C09091=1072.095,-108.990,-56.403,172.612,21.671,153.924
C09092=1072.101,-108.740,-56.412,172.614,21.673,153.924
C09093=1072.107,-108.490,-56.422,172.616,21.674,153.924
C09094=1072.114,-108.241,-56.432,172.617,21.675,153.924
C09095=1072.120,-107.991,-56.442,172.619,21.676,153.924
C09096=1072.126,-107.741,-56.451,172.621,21.677,153.924
C09097=1072.132,-107.492,-56.461,172.622,21.678,153.924
C09098=1072.138,-107.242,-56.470,172.624,21.680,153.924
C09099=1072.144,-106.992,-56.481,172.625,21.681,153.924
C09100=1072.150,-106.743,-56.491,172.626,21.681,153.924
C09101=1072.156,-106.493,-56.500,172.628,21.683,153.924
C09102=1072.162,-106.243,-56.510,172.629,21.684,153.924
C09103=1072.169,-105.993,-56.521,172.631,21.685,153.924
C09104=1072.175,-105.743,-56.531,172.633,21.686,153.924
C09105=1072.181,-105.493,-56.540,172.634,21.688,153.924
C09106=1072.187,-105.243,-56.550,172.636,21.689,153.924
C09107=1072.193,-104.994,-56.561,172.638,21.690,153.924
C09108=1072.199,-104.744,-56.570,172.639,21.691,153.924
C09109=1072.205,-104.494,-56.580,172.641,21.693,153.924
C09110=1072.212,-104.245,-56.589,172.643,21.694,153.924
C09111=1072.217,-103.995,-56.600,172.644,21.695,153.924
C09112=1072.223,-103.745,-56.610,172.646,21.696,153.924
C09113=1072.230,-103.495,-56.619,172.648,21.697,153.924
C09114=1072.236,-103.246,-56.630,172.649,21.699,153.924
C09115=1072.242,-102.996,-56.640,172.651,21.700,153.924
C09116=1072.248,-102.746,-56.649,172.652,21.701,153.924
C09117=1072.254,-102.497,-56.660,172.654,21.702,153.924
C09118=1072.260,-102.247,-56.670,172.656,21.704,153.924
C09119=1072.266,-101.997,-56.679,172.657,21.705,153.924
C09120=1072.272,-101.748,-56.690,172.659,21.706,153.924
C09121=1072.278,-101.498,-56.699,172.660,21.708,153.924
C09122=1072.284,-101.249,-56.710,172.662,21.709,153.924
C09123=1072.290,-100.999,-56.720,172.663,21.710,153.924
C09124=1072.297,-100.748,-56.730,172.664,21.711,153.924
C09125=1072.303,-100.499,-56.741,172.666,21.712,153.924
C09126=1072.309,-100.249,-56.750,172.668,21.714,153.924
C09127=1072.316,-100.000,-56.760,172.669,21.715,153.924
C09128=1072.321,-99.750,-56.771,172.671,21.716,153.924
C09129=1072.327,-99.500,-56.780,172.672,21.717,153.924
C09130=1072.334,-99.251,-56.790,172.674,21.719,153.924
C09131=1072.339,-99.001,-56.801,172.676,21.720,153.924
C09132=1072.346,-98.752,-56.811,172.677,21.721,153.924
C09133=1072.352,-98.501,-56.821,172.679,21.722,153.924
C09134=1072.359,-98.220,-56.833,172.681,21.724,153.924
C09135=1072.365,-97.938,-56.844,172.683,21.726,153.924
C09136=1072.373,-97.657,-56.855,172.685,21.727,153.924
C09137=1072.379,-97.374,-56.867,172.686,21.728,153.924
C09138=1072.386,-97.125,-56.877,172.688,21.730,153.924
C09139=1072.391,-96.875,-56.887,172.689,21.731,153.924
C09140=1072.397,-96.626,-56.898,172.691,21.733,153.924
C09141=1072.403,-96.376,-56.907,172.692,21.734,153.924
C09142=1072.409,-96.126,-56.918,172.694,21.735,153.924
C09143=1072.415,-95.877,-56.929,172.696,21.737,153.924
C09144=1072.421,-95.626,-56.939,172.697,21.738,153.924
C09145=1072.428,-95.377,-56.949,172.699,21.739,153.924
C09146=1072.433,-95.127,-56.960,172.700,21.741,153.924
C09147=1072.440,-94.878,-56.970,172.702,21.742,153.924
C09148=1072.445,-94.628,-56.980,172.703,21.744,153.924
C09149=1072.452,-94.379,-56.990,172.705,21.745,153.924
C09150=1072.457,-94.128,-57.000,172.707,21.746,153.924
C09151=1072.464,-93.879,-57.011,172.708,21.748,153.924
C09152=1072.470,-93.629,-57.022,172.710,21.749,153.924
C09153=1072.475,-93.379,-57.032,172.711,21.751,153.924
C09154=1072.482,-93.130,-57.042,172.713,21.753,153.924
C09155=1072.487,-92.880,-57.053,172.714,21.754,153.924
C09156=1072.494,-92.630,-57.063,172.716,21.755,153.924
C09157=1072.500,-92.381,-57.074,172.717,21.757,153.924
C09158=1072.506,-92.131,-57.083,172.719,21.758,153.924
C09159=1072.512,-91.881,-57.095,172.721,21.759,153.924
C09160=1072.518,-91.631,-57.105,172.722,21.761,153.924
C09161=1072.524,-91.382,-57.115,172.724,21.762,153.924
C09162=1072.530,-91.132,-57.126,172.725,21.764,153.924
C09163=1072.536,-90.882,-57.135,172.727,21.765,153.924
C09164=1072.542,-90.632,-57.147,172.728,21.766,153.924
C09165=1072.548,-90.383,-57.158,172.730,21.768,153.924
C09166=1072.554,-90.133,-57.167,172.731,21.770,153.924
C09167=1072.560,-89.883,-57.178,172.733,21.771,153.924
C09168=1072.566,-89.634,-57.188,172.735,21.773,153.924
C09169=1072.573,-89.384,-57.200,172.736,21.774,153.924
C09170=1072.578,-89.134,-57.210,172.738,21.775,153.924
C09171=1072.585,-88.885,-57.220,172.739,21.777,153.924
C09172=1072.590,-88.635,-57.231,172.741,21.778,153.924
C09173=1072.597,-88.386,-57.240,172.742,21.780,153.925
C09174=1072.603,-88.135,-57.252,172.744,21.781,153.925
C09175=1072.609,-87.886,-57.263,172.745,21.783,153.925
C09176=1072.615,-87.637,-57.273,172.747,21.784,153.925
C09177=1072.621,-87.387,-57.283,172.748,21.786,153.925
C09178=1072.628,-87.137,-57.294,172.750,21.787,153.925
C09179=1072.633,-86.887,-57.305,172.751,21.789,153.925
C09180=1072.639,-86.638,-57.315,172.753,21.790,153.925
C09181=1072.646,-86.389,-57.326,172.755,21.792,153.925
C09182=1072.652,-86.138,-57.336,172.756,21.793,153.925
C09183=1072.657,-85.888,-57.347,172.758,21.794,153.925
C09184=1072.664,-85.639,-57.357,172.759,21.796,153.925
C09185=1072.670,-85.389,-57.369,172.761,21.798,153.925
C09186=1072.676,-85.139,-57.380,172.762,21.799,153.925
C09187=1072.682,-84.890,-57.389,172.764,21.801,153.925
C09188=1072.688,-84.640,-57.400,172.765,21.802,153.925
C09189=1072.694,-84.390,-57.411,172.767,21.804,153.925
C09190=1072.701,-84.141,-57.421,172.768,21.805,153.925
C09191=1072.706,-83.891,-57.432,172.770,21.807,153.925
C09192=1072.713,-83.641,-57.444,172.772,21.808,153.925
C09193=1072.719,-83.392,-57.454,172.773,21.809,153.925
C09194=1072.725,-83.142,-57.464,172.774,21.811,153.926
C09195=1072.731,-82.892,-57.475,172.776,21.813,153.926
C09196=1072.737,-82.642,-57.486,172.778,21.814,153.926
C09197=1072.743,-82.393,-57.496,172.779,21.816,153.926
C09198=1072.750,-82.113,-57.508,172.781,21.817,153.926
C09199=1072.758,-81.834,-57.520,172.783,21.819,153.926
C09200=1072.764,-81.554,-57.533,172.784,21.821,153.926
C09201=1072.771,-81.275,-57.545,172.786,21.823,153.926
C09202=1072.777,-81.026,-57.556,172.788,21.824,153.926
C09203=1072.784,-80.776,-57.566,172.789,21.826,153.926
C09204=1072.790,-80.526,-57.577,172.791,21.827,153.926
C09205=1072.795,-80.277,-57.588,172.792,21.829,153.926
C09206=1072.802,-80.027,-57.599,172.793,21.831,153.926
C09207=1072.808,-79.778,-57.610,172.795,21.832,153.926
C09208=1072.814,-79.527,-57.620,172.797,21.833,153.926
C09209=1072.820,-79.277,-57.631,172.798,21.835,153.926
C09210=1072.826,-79.028,-57.642,172.800,21.837,153.926
C09211=1072.832,-78.778,-57.653,172.801,21.839,153.927
C09212=1072.838,-78.528,-57.664,172.803,21.840,153.927
C09213=1072.844,-78.279,-57.675,172.804,21.842,153.927
C09214=1072.850,-78.030,-57.687,172.805,21.843,153.927
C09215=1072.857,-77.780,-57.697,172.807,21.845,153.927
C09216=1072.862,-77.530,-57.708,172.809,21.847,153.927
C09217=1072.869,-77.280,-57.719,172.811,21.848,153.927
C09218=1072.875,-77.031,-57.730,172.812,21.850,153.927
C09219=1072.880,-76.781,-57.741,172.814,21.852,153.927
C09220=1072.887,-76.531,-57.752,172.815,21.854,153.927
C09221=1072.892,-76.281,-57.763,172.817,21.855,153.927
C09222=1072.898,-76.032,-57.774,172.818,21.857,153.927
C09223=1072.904,-75.782,-57.785,172.820,21.858,153.927
C09224=1072.910,-75.532,-57.796,172.821,21.860,153.928
C09225=1072.917,-75.282,-57.807,172.823,21.862,153.928
C09226=1072.923,-75.033,-57.818,172.824,21.864,153.928
C09227=1072.929,-74.783,-57.829,172.826,21.865,153.928
C09228=1072.935,-74.534,-57.841,172.827,21.867,153.928
C09229=1072.941,-74.284,-57.851,172.829,21.868,153.928
C09230=1072.947,-74.034,-57.863,172.830,21.870,153.928
C09231=1072.953,-73.785,-57.874,172.832,21.872,153.928
C09232=1072.959,-73.535,-57.884,172.833,21.874,153.928
C09233=1072.965,-73.285,-57.896,172.835,21.875,153.928
C09234=1072.970,-73.035,-57.907,172.836,21.877,153.928
C09235=1072.976,-72.786,-57.919,172.837,21.879,153.929
C09236=1072.983,-72.536,-57.930,172.839,21.880,153.929
C09237=1072.988,-72.287,-57.941,172.840,21.882,153.929
C09238=1072.994,-72.037,-57.952,172.842,21.884,153.929
C09239=1073.000,-71.787,-57.963,172.843,21.886,153.929
C09240=1073.007,-71.538,-57.975,172.845,21.888,153.929
C09241=1073.012,-71.288,-57.986,172.847,21.890,153.929
C09242=1073.018,-71.038,-57.997,172.848,21.891,153.929
C09243=1073.024,-70.789,-58.008,172.850,21.893,153.929
C09244=1073.030,-70.538,-58.019,172.851,21.895,153.930
C09245=1073.036,-70.290,-58.031,172.853,21.897,153.930
C09246=1073.042,-70.039,-58.042,172.854,21.898,153.930
C09247=1073.048,-69.790,-58.053,172.856,21.900,153.930
C09248=1073.053,-69.540,-58.065,172.857,21.902,153.930
C09249=1073.060,-69.291,-58.077,172.859,21.904,153.930
C09250=1073.065,-69.041,-58.087,172.860,21.906,153.930
C09251=1073.072,-68.791,-58.099,172.861,21.908,153.930
C09252=1073.078,-68.542,-58.110,172.863,21.909,153.930
C09253=1073.084,-68.292,-58.122,172.864,21.911,153.930
C09254=1073.089,-68.042,-58.133,172.866,21.913,153.931
C09255=1073.095,-67.792,-58.144,172.867,21.914,153.931
C09256=1073.102,-67.543,-58.156,172.869,21.916,153.931
C09257=1073.107,-67.293,-58.167,172.870,21.918,153.931
C09258=1073.114,-67.043,-58.178,172.871,21.920,153.931
C09259=1073.119,-66.794,-58.190,172.873,21.921,153.931
C09260=1073.125,-66.544,-58.201,172.875,21.924,153.931
C09261=1073.131,-66.295,-58.213,172.877,21.926,153.931
C09262=1073.138,-66.018,-58.226,172.878,21.928,153.932
C09263=1073.145,-65.740,-58.238,172.879,21.930,153.932
C09264=1073.152,-65.463,-58.250,172.881,21.931,153.932
C09265=1073.158,-65.185,-58.264,172.883,21.934,153.932
C09266=1073.164,-64.937,-58.275,172.885,21.935,153.932
C09267=1073.170,-64.686,-58.286,172.886,21.937,153.932
C09268=1073.176,-64.438,-58.298,172.887,21.939,153.932
C09269=1073.182,-64.187,-58.310,172.889,21.941,153.932
C09270=1073.188,-63.937,-58.321,172.890,21.943,153.933
C09271=1073.194,-63.688,-58.333,172.892,21.944,153.933
C09272=1073.200,-63.438,-58.344,172.893,21.946,153.933
C09273=1073.206,-63.189,-58.356,172.895,21.948,153.933
C09274=1073.212,-62.938,-58.367,172.896,21.950,153.933
C09275=1073.218,-62.689,-58.379,172.897,21.952,153.933
C09276=1073.224,-62.439,-58.390,172.899,21.953,153.933
C09277=1073.230,-62.190,-58.402,172.900,21.955,153.933
C09278=1073.236,-61.940,-58.414,172.903,21.958,153.933
C09279=1073.242,-61.691,-58.425,172.904,21.960,153.934
C09280=1073.248,-61.441,-58.436,172.905,21.962,153.934
C09281=1073.254,-61.192,-58.448,172.907,21.963,153.934
C09282=1073.260,-60.941,-58.460,172.908,21.965,153.934
C09283=1073.267,-60.692,-58.472,172.910,21.967,153.934
C09284=1073.272,-60.442,-58.483,172.911,21.969,153.934
C09285=1073.279,-60.193,-58.495,172.912,21.971,153.934
C09286=1073.284,-59.943,-58.506,172.914,21.973,153.935
C09287=1073.291,-59.693,-58.518,172.915,21.974,153.935
C09288=1073.297,-59.443,-58.529,172.917,21.976,153.935
C09289=1073.302,-59.194,-58.542,172.918,21.978,153.935
C09290=1073.309,-58.944,-58.553,172.920,21.980,153.935
C09291=1073.315,-58.695,-58.564,172.921,21.982,153.935
C09292=1073.321,-58.445,-58.576,172.923,21.984,153.935
C09293=1073.327,-58.195,-58.588,172.925,21.986,153.935
C09294=1073.333,-57.946,-58.600,172.926,21.987,153.935
C09295=1073.339,-57.696,-58.611,172.928,21.989,153.936
C09296=1073.345,-57.446,-58.624,172.929,21.991,153.936
C09297=1073.351,-57.197,-58.635,172.930,21.993,153.936
C09298=1073.358,-56.947,-58.646,172.932,21.995,153.936
C09299=1073.363,-56.698,-58.659,172.933,21.997,153.936
C09300=1073.369,-56.448,-58.670,172.935,21.999,153.936
C09301=1073.376,-56.198,-58.682,172.936,22.001,153.937
C09302=1073.382,-55.949,-58.693,172.937,22.002,153.937
C09303=1073.388,-55.699,-58.705,172.939,22.004,153.937
C09304=1073.394,-55.449,-58.717,172.940,22.006,153.937
C09305=1073.400,-55.200,-58.729,172.942,22.008,153.937
C09306=1073.406,-54.950,-58.741,172.944,22.010,153.937
C09307=1073.413,-54.700,-58.753,172.945,22.012,153.937
C09308=1073.419,-54.451,-58.764,172.947,22.014,153.937
C09309=1073.425,-54.201,-58.777,172.948,22.016,153.938
C09310=1073.431,-53.951,-58.788,172.949,22.018,153.938
C09311=1073.438,-53.702,-58.800,172.951,22.020,153.938
C09312=1073.443,-53.452,-58.812,172.952,22.022,153.938
C09313=1073.449,-53.202,-58.823,172.954,22.024,153.938
C09314=1073.456,-52.953,-58.835,172.955,22.025,153.938
C09315=1073.461,-52.703,-58.847,172.957,22.027,153.938
C09316=1073.468,-52.454,-58.859,172.958,22.029,153.939
C09317=1073.473,-52.203,-58.871,172.959,22.031,153.939
C09318=1073.480,-51.954,-58.883,172.962,22.033,153.939
C09319=1073.486,-51.705,-58.895,172.963,22.035,153.939
C09320=1073.492,-51.455,-58.907,172.964,22.037,153.939
C09321=1073.499,-51.206,-58.919,172.966,22.039,153.939
C09322=1073.505,-50.955,-58.931,172.967,22.041,153.939
C09323=1073.510,-50.706,-58.943,172.969,22.043,153.940
C09324=1073.517,-50.457,-58.955,172.970,22.045,153.940
C09325=1073.523,-50.207,-58.967,172.971,22.047,153.940
C09326=1073.529,-49.931,-58.980,172.973,22.049,153.940
C09327=1073.536,-49.655,-58.994,172.975,22.052,153.940
C09328=1073.543,-49.379,-59.007,172.976,22.054,153.940
C09329=1073.549,-49.103,-59.021,172.978,22.056,153.941
C09330=1073.555,-48.854,-59.033,172.979,22.058,153.941
C09331=1073.561,-48.604,-59.044,172.981,22.060,153.941
C09332=1073.567,-48.354,-59.056,172.983,22.062,153.941
C09333=1073.573,-48.105,-59.069,172.984,22.064,153.941
C09334=1073.579,-47.855,-59.081,172.985,22.066,153.941
C09335=1073.585,-47.605,-59.093,172.987,22.068,153.942
C09336=1073.591,-47.356,-59.106,172.988,22.070,153.942
C09337=1073.597,-47.106,-59.118,172.989,22.072,153.942
C09338=1073.603,-46.857,-59.130,172.991,22.074,153.942
C09339=1073.609,-46.607,-59.142,172.992,22.076,153.942
C09340=1073.614,-46.358,-59.155,172.993,22.078,153.942
C09341=1073.621,-46.108,-59.167,172.995,22.080,153.943
C09342=1073.627,-45.858,-59.179,172.997,22.083,153.943
C09343=1073.633,-45.608,-59.191,172.998,22.085,153.943
C09344=1073.639,-45.359,-59.203,173.000,22.087,153.943
C09345=1073.644,-45.109,-59.215,173.001,22.089,153.943
C09346=1073.650,-44.859,-59.228,173.003,22.091,153.943
C09347=1073.657,-44.610,-59.240,173.004,22.093,153.944
C09348=1073.662,-44.360,-59.252,173.005,22.095,153.944
C09349=1073.668,-44.111,-59.264,173.007,22.097,153.944
C09350=1073.675,-43.861,-59.276,173.008,22.099,153.944
C09351=1073.681,-43.611,-59.289,173.009,22.101,153.944
C09352=1073.687,-43.361,-59.301,173.012,22.103,153.944
C09353=1073.692,-43.112,-59.314,173.013,22.106,153.945
C09354=1073.699,-42.862,-59.326,173.014,22.108,153.945
C09355=1073.705,-42.613,-59.339,173.016,22.110,153.945
C09356=1073.711,-42.363,-59.351,173.017,22.112,153.945
C09357=1073.717,-42.114,-59.363,173.018,22.113,153.945
C09358=1073.723,-41.865,-59.376,173.020,22.116,153.946
C09359=1073.729,-41.615,-59.388,173.021,22.118,153.946
C09360=1073.735,-41.365,-59.401,173.022,22.120,153.946
C09361=1073.741,-41.115,-59.413,173.024,22.122,153.946
C09362=1073.747,-40.865,-59.425,173.026,22.124,153.946
C09363=1073.752,-40.616,-59.437,173.027,22.126,153.947
C09364=1073.759,-40.367,-59.449,173.029,22.128,153.947
C09365=1073.765,-40.117,-59.462,173.030,22.130,153.947
C09366=1073.771,-39.867,-59.475,173.031,22.132,153.947
C09367=1073.777,-39.618,-59.488,173.033,22.135,153.947
C09368=1073.784,-39.368,-59.500,173.034,22.137,153.947
C09369=1073.790,-39.118,-59.512,173.035,22.139,153.948
C09370=1073.795,-38.869,-59.524,173.037,22.140,153.948
C09371=1073.801,-38.619,-59.537,173.038,22.143,153.948
C09372=1073.807,-38.369,-59.549,173.040,22.145,153.948
C09373=1073.814,-38.120,-59.562,173.042,22.147,153.948
C09374=1073.820,-37.870,-59.575,173.043,22.150,153.949
C09375=1073.826,-37.620,-59.587,173.044,22.152,153.949
C09376=1073.831,-37.371,-59.599,173.046,22.154,153.949
C09377=1073.837,-37.121,-59.612,173.047,22.156,153.949
C09378=1073.843,-36.872,-59.625,173.048,22.158,153.949
C09379=1073.849,-36.622,-59.638,173.050,22.160,153.949
C09380=1073.855,-36.372,-59.650,173.051,22.162,153.950
C09381=1073.861,-36.122,-59.663,173.053,22.165,153.950
C09382=1073.866,-35.873,-59.675,173.054,22.167,153.950
C09383=1073.872,-35.624,-59.688,173.056,22.169,153.950
C09384=1073.878,-35.374,-59.701,173.057,22.171,153.950
C09385=1073.884,-35.124,-59.713,173.058,22.173,153.951
C09386=1073.890,-34.875,-59.727,173.060,22.175,153.951
C09387=1073.896,-34.625,-59.739,173.061,22.177,153.951
C09388=1073.903,-34.375,-59.751,173.062,22.180,153.951
C09389=1073.909,-34.126,-59.764,173.064,22.182,153.951
C09390=1073.915,-33.851,-59.779,173.066,22.185,153.952
C09391=1073.922,-33.575,-59.792,173.067,22.186,153.952
C09392=1073.928,-33.300,-59.806,173.068,22.189,153.952
C09393=1073.935,-33.024,-59.820,173.071,22.192,153.952
C09394=1073.941,-32.775,-59.833,173.072,22.194,153.953
C09395=1073.947,-32.525,-59.846,173.073,22.196,153.953
C09396=1073.953,-32.275,-59.858,173.075,22.198,153.953
C09397=1073.959,-32.026,-59.872,173.076,22.200,153.953
C09398=1073.965,-31.776,-59.884,173.077,22.203,153.953
C09399=1073.971,-31.526,-59.897,173.079,22.204,153.954
C09400=1073.977,-31.277,-59.910,173.081,22.207,153.954
C09401=1073.983,-31.027,-59.923,173.082,22.209,153.954
C09402=1073.989,-30.777,-59.935,173.083,22.211,153.954
C09403=1073.995,-30.528,-59.948,173.085,22.214,153.954
C09404=1074.001,-30.278,-59.961,173.086,22.216,153.955
C09405=1074.007,-30.029,-59.974,173.087,22.218,153.955
C09406=1074.013,-29.779,-59.987,173.089,22.220,153.955
C09407=1074.019,-29.530,-60.000,173.090,22.222,153.955
C09408=1074.024,-29.280,-60.012,173.091,22.224,153.955
C09409=1074.030,-29.030,-60.025,173.094,22.227,153.956
C09410=1074.037,-28.781,-60.038,173.095,22.229,153.956
C09411=1074.042,-28.531,-60.051,173.096,22.231,153.956
C09412=1074.049,-28.282,-60.064,173.097,22.233,153.956
C09413=1074.055,-28.032,-60.076,173.099,22.235,153.956
C09414=1074.061,-27.783,-60.090,173.100,22.238,153.957
C09415=1074.067,-27.533,-60.102,173.101,22.240,153.957
C09416=1074.073,-27.284,-60.115,173.103,22.242,153.957
C09417=1074.079,-27.034,-60.128,173.104,22.244,153.957
C09418=1074.084,-26.784,-60.142,173.106,22.246,153.957
C09419=1074.090,-26.534,-60.154,173.108,22.249,153.958
C09420=1074.096,-26.285,-60.168,173.109,22.251,153.958
C09421=1074.102,-26.035,-60.180,173.110,22.253,153.958
C09422=1074.109,-25.786,-60.194,173.111,22.256,153.958
C09423=1074.114,-25.536,-60.207,173.113,22.258,153.959
C09424=1074.120,-25.287,-60.220,173.114,22.260,153.959
C09425=1074.126,-25.037,-60.233,173.115,22.262,153.959
C09426=1074.132,-24.787,-60.246,173.117,22.265,153.959
C09427=1074.138,-24.538,-60.260,173.119,22.267,153.959
C09428=1074.143,-24.288,-60.272,173.120,22.269,153.960
C09429=1074.150,-24.039,-60.285,173.121,22.272,153.960
C09430=1074.156,-23.789,-60.299,173.123,22.274,153.960
C09431=1074.162,-23.540,-60.311,173.124,22.276,153.960
C09432=1074.167,-23.290,-60.325,173.125,22.278,153.961
C09433=1074.173,-23.040,-60.338,173.127,22.281,153.961
C09434=1074.179,-22.791,-60.351,173.129,22.283,153.961
C09435=1074.186,-22.542,-60.364,173.130,22.285,153.961
C09436=1074.191,-22.291,-60.377,173.131,22.288,153.962
C09437=1074.197,-22.042,-60.391,173.133,22.290,153.962
C09438=1074.203,-21.793,-60.404,173.134,22.292,153.962
C09439=1074.208,-21.543,-60.417,173.135,22.294,153.962
C09440=1074.215,-21.293,-60.431,173.137,22.297,153.963
C09441=1074.221,-21.043,-60.444,173.138,22.298,153.963
C09442=1074.227,-20.794,-60.457,173.140,22.301,153.963
C09443=1074.233,-20.544,-60.470,173.141,22.304,153.963
C09444=1074.239,-20.295,-60.484,173.143,22.306,153.963
C09445=1074.245,-20.045,-60.496,173.144,22.308,153.964
C09446=1074.251,-19.796,-60.509,173.145,22.310,153.964
C09447=1074.257,-19.546,-60.523,173.146,22.313,153.964
C09448=1074.263,-19.297,-60.537,173.148,22.315,153.964
C09449=1074.269,-19.047,-60.549,173.149,22.317,153.965
C09450=1074.274,-18.797,-60.563,173.151,22.320,153.965
C09451=1074.280,-18.548,-60.576,173.153,22.322,153.965
C09452=1074.287,-18.299,-60.590,173.154,22.324,153.965
C09453=1074.292,-18.048,-60.603,173.155,22.327,153.965
C09454=1074.299,-17.772,-60.618,173.156,22.329,153.966
C09455=1074.306,-17.496,-60.633,173.159,22.331,153.966
C09456=1074.313,-17.219,-60.647,173.160,22.334,153.966
C09457=1074.319,-16.943,-60.662,173.161,22.336,153.966
C09458=1074.325,-16.694,-60.675,173.162,22.339,153.967
C09459=1074.331,-16.444,-60.689,173.165,22.341,153.967
C09460=1074.337,-16.195,-60.702,173.166,22.344,153.967
C09461=1074.343,-15.946,-60.716,173.167,22.346,153.967
C09462=1074.349,-15.695,-60.730,173.168,22.348,153.968
C09463=1074.355,-15.445,-60.742,173.170,22.350,153.968
C09464=1074.362,-15.196,-60.756,173.171,22.352,153.968
C09465=1074.367,-14.947,-60.769,173.172,22.355,153.968
C09466=1074.373,-14.697,-60.783,173.174,22.358,153.969
C09467=1074.379,-14.448,-60.797,173.176,22.360,153.969
C09468=1074.385,-14.198,-60.810,173.177,22.362,153.969
C09469=1074.390,-13.949,-60.824,173.178,22.364,153.969
C09470=1074.397,-13.699,-60.837,173.179,22.367,153.970
C09471=1074.403,-13.449,-60.851,173.181,22.369,153.970
C09472=1074.409,-13.199,-60.864,173.182,22.371,153.970
C09473=1074.414,-12.950,-60.878,173.183,22.374,153.970
C09474=1074.420,-12.701,-60.891,173.185,22.377,153.971
C09475=1074.426,-12.451,-60.905,173.187,22.379,153.971
C09476=1074.432,-12.202,-60.918,173.188,22.381,153.971
C09477=1074.438,-11.952,-60.932,173.189,22.383,153.971
C09478=1074.444,-11.702,-60.946,173.191,22.385,153.971
C09479=1074.450,-11.453,-60.959,173.192,22.388,153.972
C09480=1074.455,-11.203,-60.973,173.193,22.390,153.972
C09481=1074.461,-10.954,-60.987,173.195,22.393,153.972
C09482=1074.467,-10.704,-61.000,173.197,22.395,153.972
C09483=1074.474,-10.454,-61.014,173.198,22.397,153.973
C09484=1074.479,-10.205,-61.028,173.199,22.400,153.973
C09485=1074.485,-9.955,-61.041,173.200,22.402,153.973
C09486=1074.491,-9.706,-61.055,173.202,22.404,153.973
C09487=1074.497,-9.457,-61.068,173.203,22.407,153.974
C09488=1074.503,-9.206,-61.083,173.204,22.409,153.974
C09489=1074.509,-8.957,-61.096,173.206,22.412,153.974
C09490=1074.515,-8.708,-61.110,173.208,22.414,153.974
C09491=1074.520,-8.458,-61.124,173.209,22.416,153.975
C09492=1074.527,-8.209,-61.137,173.210,22.419,153.975
C09493=1074.533,-7.959,-61.152,173.211,22.421,153.975
C09494=1074.539,-7.710,-61.165,173.213,22.423,153.975
C09495=1074.545,-7.460,-61.179,173.214,22.426,153.976
C09496=1074.550,-7.211,-61.193,173.216,22.429,153.976
C09497=1074.557,-6.961,-61.206,173.217,22.431,153.976
C09498=1074.562,-6.711,-61.220,173.219,22.433,153.976
C09499=1074.569,-6.462,-61.234,173.220,22.435,153.977
C09500=1074.574,-6.212,-61.247,173.221,22.438,153.977
C09501=1074.580,-5.962,-61.262,173.223,22.440,153.977
C09502=1074.587,-5.713,-61.276,173.224,22.442,153.977
C09503=1074.592,-5.464,-61.289,173.226,22.445,153.978
C09504=1074.598,-5.214,-61.303,173.227,22.447,153.978
C09505=1074.604,-4.964,-61.317,173.228,22.449,153.978
C09506=1074.610,-4.715,-61.331,173.230,22.452,153.978
C09507=1074.616,-4.465,-61.344,173.231,22.454,153.979
C09508=1074.623,-4.216,-61.359,173.232,22.457,153.979
C09509=1074.629,-3.966,-61.372,173.234,22.459,153.979
C09510=1074.634,-3.717,-61.386,173.236,22.461,153.979
C09511=1074.640,-3.467,-61.400,173.237,22.464,153.980
C09512=1074.647,-3.217,-61.414,173.238,22.466,153.980
C09513=1074.652,-2.968,-61.428,173.239,22.469,153.980
C09514=1074.658,-2.719,-61.442,173.241,22.471,153.981
C09515=1074.664,-2.468,-61.456,173.242,22.473,153.981
C09516=1074.669,-2.219,-61.470,173.243,22.476,153.981
C09517=1074.675,-1.970,-61.485,173.245,22.479,153.981
C09518=1074.681,-1.692,-61.500,173.247,22.481,153.982
C09519=1074.688,-1.414,-61.515,173.248,22.484,153.982
C09520=1074.694,-1.136,-61.531,173.250,22.487,153.982
C09521=1074.701,-0.858,-61.547,173.251,22.489,153.982
C09522=1074.707,-0.608,-61.561,173.252,22.492,153.983
C09523=1074.712,-0.359,-61.576,173.253,22.494,153.983
C09524=1074.719,-0.109,-61.589,173.256,22.497,153.983
C09525=1074.725,0.140,-61.603,173.257,22.499,153.984
C09526=1074.730,0.390,-61.617,173.258,22.502,153.984
C09527=1074.737,0.639,-61.632,173.259,22.504,153.984
C09528=1074.742,0.889,-61.646,173.261,22.506,153.984
C09529=1074.748,1.138,-61.661,173.262,22.509,153.985
C09530=1074.753,1.387,-61.674,173.263,22.511,153.985
C09531=1074.759,1.638,-61.689,173.265,22.514,153.985
C09532=1074.765,1.887,-61.703,173.266,22.516,153.985
C09533=1074.771,2.136,-61.717,173.268,22.519,153.986
C09534=1074.777,2.386,-61.731,173.269,22.521,153.986
C09535=1074.783,2.635,-61.745,173.270,22.524,153.986
C09536=1074.789,2.885,-61.759,173.272,22.526,153.986
C09537=1074.795,3.134,-61.774,173.273,22.528,153.987
C09538=1074.801,3.384,-61.788,173.275,22.531,153.987
C09539=1074.806,3.633,-61.803,173.276,22.533,153.987
C09540=1074.812,3.883,-61.817,173.277,22.536,153.988
C09541=1074.818,4.133,-61.831,173.279,22.538,153.988
C09542=1074.824,4.382,-61.845,173.280,22.541,153.988
C09543=1074.830,4.632,-61.859,173.281,22.543,153.988
C09544=1074.836,4.881,-61.874,173.282,22.546,153.989
C09545=1074.842,5.131,-61.888,173.284,22.549,153.989
C09546=1074.847,5.380,-61.903,173.286,22.550,153.989
C09547=1074.854,5.629,-61.916,173.287,22.553,153.989
C09548=1074.860,5.879,-61.931,173.288,22.555,153.990
C09549=1074.866,6.129,-61.945,173.290,22.558,153.990
C09550=1074.872,6.378,-61.960,173.291,22.560,153.990
C09551=1074.877,6.628,-61.974,173.293,22.563,153.991
C09552=1074.883,6.877,-61.988,173.294,22.566,153.991
C09553=1074.889,7.127,-62.003,173.295,22.568,153.991
C09554=1074.895,7.376,-62.017,173.297,22.570,153.991
C09555=1074.901,7.626,-62.031,173.298,22.572,153.992
C09556=1074.907,7.875,-62.046,173.299,22.575,153.992
C09557=1074.913,8.124,-62.060,173.301,22.577,153.992
C09558=1074.919,8.375,-62.075,173.303,22.580,153.992
C09559=1074.925,8.624,-62.089,173.304,22.582,153.993
C09560=1074.931,8.874,-62.104,173.305,22.585,153.993
C09561=1074.936,9.123,-62.118,173.306,22.587,153.993
C09562=1074.943,9.372,-62.133,173.308,22.590,153.994
C09563=1074.948,9.622,-62.147,173.309,22.592,153.994
C09564=1074.955,9.872,-62.162,173.310,22.594,153.994
C09565=1074.960,10.121,-62.176,173.312,22.597,153.994
C09566=1074.966,10.371,-62.191,173.314,22.599,153.994
C09567=1074.972,10.620,-62.205,173.315,22.602,153.995
C09568=1074.978,10.870,-62.219,173.316,22.604,153.995
C09569=1074.984,11.119,-62.234,173.317,22.607,153.995
C09570=1074.990,11.369,-62.249,173.319,22.609,153.996
C09571=1074.996,11.618,-62.263,173.321,22.612,153.996
C09572=1075.002,11.868,-62.278,173.322,22.615,153.996
C09573=1075.008,12.117,-62.292,173.323,22.616,153.996
C09574=1075.014,12.367,-62.307,173.325,22.619,153.997
C09575=1075.020,12.616,-62.321,173.326,22.621,153.997
C09576=1075.026,12.866,-62.336,173.327,22.624,153.997
C09577=1075.032,13.115,-62.351,173.329,22.627,153.997
C09578=1075.038,13.365,-62.365,173.330,22.629,153.998
C09579=1075.044,13.614,-62.380,173.332,22.631,153.998
C09580=1075.050,13.864,-62.394,173.333,22.634,153.998
C09581=1075.056,14.113,-62.409,173.334,22.636,153.998
C09582=1075.063,14.393,-62.426,173.336,22.639,153.999
C09583=1075.069,14.673,-62.442,173.338,22.642,153.999
C09584=1075.076,14.953,-62.458,173.339,22.644,153.999
C09585=1075.082,15.233,-62.475,173.341,22.647,154.000
C09586=1075.088,15.483,-62.490,173.342,22.650,154.000
C09587=1075.094,15.732,-62.504,173.343,22.652,154.000
C09588=1075.100,15.981,-62.519,173.344,22.655,154.001
C09589=1075.106,16.230,-62.534,173.346,22.657,154.001
C09590=1075.112,16.481,-62.549,173.348,22.660,154.001
C09591=1075.117,16.730,-62.563,173.349,22.662,154.002
C09592=1075.124,16.979,-62.578,173.350,22.665,154.002
C09593=1075.129,17.228,-62.593,173.352,22.667,154.002
C09594=1075.135,17.478,-62.608,173.353,22.670,154.002
C09595=1075.141,17.727,-62.623,173.354,22.672,154.003
C09596=1075.147,17.977,-62.638,173.356,22.675,154.003
C09597=1075.153,18.227,-62.652,173.358,22.677,154.003
C09598=1075.158,18.477,-62.667,173.359,22.679,154.003
C09599=1075.165,18.726,-62.682,173.360,22.682,154.004
C09600=1075.171,18.975,-62.697,173.361,22.684,154.004
C09601=1075.177,19.225,-62.712,173.363,22.687,154.004
C09602=1075.182,19.474,-62.727,173.365,22.690,154.004
C09603=1075.188,19.724,-62.742,173.366,22.692,154.005
C09604=1075.194,19.973,-62.757,173.367,22.694,154.005
C09605=1075.200,20.223,-62.772,173.368,22.697,154.005
C09606=1075.206,20.472,-62.787,173.370,22.699,154.006
C09607=1075.212,20.721,-62.802,173.371,22.702,154.006
C09608=1075.218,20.971,-62.817,173.373,22.705,154.006
C09609=1075.223,21.220,-62.832,173.374,22.707,154.006
C09610=1075.230,21.470,-62.847,173.376,22.709,154.007
C09611=1075.235,21.719,-62.862,173.377,22.712,154.007
C09612=1075.241,21.969,-62.877,173.378,22.714,154.007
C09613=1075.247,22.219,-62.892,173.379,22.717,154.008
C09614=1075.253,22.468,-62.907,173.381,22.720,154.008
C09615=1075.259,22.717,-62.922,173.383,22.722,154.008
C09616=1075.264,22.967,-62.937,173.384,22.724,154.008
C09617=1075.270,23.216,-62.952,173.385,22.727,154.009
C09618=1075.277,23.466,-62.967,173.386,22.729,154.009
C09619=1075.282,23.715,-62.982,173.388,22.732,154.009
C09620=1075.288,23.965,-62.997,173.390,22.735,154.010
C09621=1075.293,24.214,-63.012,173.391,22.737,154.010
C09622=1075.300,24.464,-63.027,173.392,22.739,154.010
C09623=1075.305,24.714,-63.043,173.394,22.742,154.010
C09624=1075.311,24.963,-63.057,173.395,22.744,154.011
C09625=1075.317,25.212,-63.072,173.397,22.747,154.011
C09626=1075.323,25.462,-63.088,173.398,22.750,154.011
C09627=1075.329,25.711,-63.103,173.399,22.752,154.012
C09628=1075.335,25.961,-63.119,173.401,22.754,154.012
C09629=1075.341,26.210,-63.134,173.402,22.757,154.012
C09630=1075.347,26.459,-63.148,173.403,22.759,154.012
C09631=1075.353,26.709,-63.164,173.405,22.762,154.013
C09632=1075.359,26.959,-63.179,173.407,22.765,154.013
C09633=1075.364,27.208,-63.194,173.408,22.767,154.013
C09634=1075.371,27.457,-63.210,173.409,22.769,154.014
C09635=1075.376,27.707,-63.225,173.410,22.772,154.014
C09636=1075.382,27.956,-63.240,173.412,22.774,154.014
C09637=1075.388,28.206,-63.255,173.414,22.777,154.014
C09638=1075.394,28.456,-63.270,173.415,22.780,154.015
C09639=1075.400,28.704,-63.286,173.416,22.782,154.015
C09640=1075.406,28.954,-63.301,173.417,22.784,154.015
C09641=1075.412,29.204,-63.317,173.418,22.787,154.016
C09642=1075.417,29.453,-63.332,173.421,22.790,154.016
C09643=1075.423,29.702,-63.347,173.422,22.793,154.016
C09644=1075.429,29.952,-63.363,173.423,22.795,154.016
C09645=1075.435,30.201,-63.377,173.424,22.798,154.017
C09646=1075.441,30.483,-63.395,173.427,22.800,154.017
C09647=1075.448,30.764,-63.413,173.428,22.803,154.017
C09648=1075.455,31.045,-63.430,173.429,22.806,154.018
C09649=1075.460,31.326,-63.448,173.431,22.809,154.018
C09650=1075.467,31.576,-63.463,173.432,22.812,154.018
C09651=1075.473,31.826,-63.478,173.433,22.814,154.019
C09652=1075.479,32.075,-63.494,173.435,22.816,154.019
C09653=1075.484,32.324,-63.509,173.437,22.819,154.019
C09654=1075.490,32.574,-63.524,173.438,22.822,154.020
C09655=1075.497,32.823,-63.540,173.439,22.824,154.020
C09656=1075.502,33.073,-63.555,173.440,22.827,154.020
C09657=1075.507,33.323,-63.571,173.442,22.829,154.020
C09658=1075.514,33.572,-63.586,173.444,22.832,154.021
C09659=1075.520,33.822,-63.602,173.445,22.834,154.021
C09660=1075.525,34.070,-63.618,173.446,22.837,154.021
C09661=1075.531,34.320,-63.633,173.448,22.839,154.022
C09662=1075.537,34.570,-63.648,173.449,22.842,154.022
C09663=1075.543,34.819,-63.665,173.451,22.844,154.022
C09664=1075.549,35.068,-63.679,173.452,22.847,154.022
C09665=1075.555,35.318,-63.695,173.454,22.849,154.023
C09666=1075.560,35.568,-63.711,173.455,22.852,154.023
C09667=1075.567,35.817,-63.726,173.456,22.854,154.023
C09668=1075.572,36.066,-63.742,173.458,22.857,154.023
C09669=1075.578,36.316,-63.757,173.459,22.859,154.024
C09670=1075.584,36.565,-63.773,173.461,22.862,154.024
C09671=1075.590,36.815,-63.789,173.462,22.864,154.024
C09672=1075.596,37.064,-63.805,173.463,22.867,154.025
C09673=1075.601,37.313,-63.820,173.464,22.869,154.025
C09674=1075.608,37.562,-63.836,173.467,22.872,154.025
C09675=1075.613,37.812,-63.851,173.468,22.874,154.025
C09676=1075.619,38.062,-63.868,173.469,22.877,154.026
C09677=1075.625,38.312,-63.883,173.470,22.880,154.026
C09678=1075.631,38.560,-63.898,173.471,22.882,154.026
C09679=1075.637,38.810,-63.914,173.474,22.885,154.027
C09680=1075.643,39.059,-63.930,173.475,22.887,154.027
C09681=1075.648,39.309,-63.946,173.476,22.890,154.027
C09682=1075.654,39.559,-63.962,173.477,22.892,154.028
C09683=1075.659,39.808,-63.977,173.479,22.895,154.028
C09684=1075.665,40.057,-63.993,173.481,22.897,154.028
C09685=1075.672,40.306,-64.009,173.482,22.900,154.028
C09686=1075.678,40.556,-64.025,173.483,22.902,154.029
C09687=1075.683,40.806,-64.041,173.485,22.905,154.029
C09688=1075.689,41.055,-64.056,173.486,22.908,154.029
C09689=1075.694,41.304,-64.072,173.488,22.910,154.030
C09690=1075.700,41.554,-64.089,173.489,22.913,154.030
C09691=1075.706,41.804,-64.104,173.490,22.915,154.030
C09692=1075.712,42.053,-64.120,173.492,22.918,154.031
C09693=1075.718,42.302,-64.137,173.493,22.920,154.031
C09694=1075.724,42.551,-64.151,173.495,22.923,154.031
C09695=1075.730,42.801,-64.167,173.496,22.925,154.031
C09696=1075.735,43.051,-64.183,173.498,22.928,154.032
C09697=1075.741,43.300,-64.199,173.499,22.930,154.032
C09698=1075.747,43.549,-64.215,173.500,22.933,154.032
C09699=1075.753,43.799,-64.232,173.502,22.936,154.032
C09700=1075.759,44.049,-64.247,173.503,22.938,154.033
C09701=1075.764,44.297,-64.263,173.505,22.941,154.033
C09702=1075.770,44.547,-64.279,173.506,22.943,154.033
C09703=1075.776,44.797,-64.295,173.508,22.946,154.034
C09704=1075.782,45.046,-64.311,173.509,22.949,154.034
C09705=1075.788,45.295,-64.327,173.511,22.951,154.034
C09706=1075.792,45.544,-64.344,173.512,22.953,154.035
C09707=1075.798,45.794,-64.359,173.513,22.956,154.035
C09708=1075.804,46.044,-64.376,173.515,22.959,154.035
C09709=1075.810,46.293,-64.392,173.516,22.962,154.036
C09710=1075.816,46.575,-64.410,173.518,22.964,154.036
C09711=1075.822,46.855,-64.428,173.520,22.967,154.036
C09712=1075.829,47.137,-64.446,173.521,22.970,154.037
C09713=1075.836,47.418,-64.465,173.523,22.973,154.037
C09714=1075.841,47.668,-64.481,173.524,22.976,154.037
C09715=1075.847,47.918,-64.497,173.525,22.978,154.037
C09716=1075.853,48.167,-64.513,173.527,22.980,154.038
C09717=1075.858,48.415,-64.529,173.529,22.983,154.038
C09718=1075.864,48.665,-64.545,173.530,22.986,154.038
C09719=1075.870,48.914,-64.562,173.531,22.989,154.039
C09720=1075.876,49.164,-64.578,173.532,22.991,154.039
C09721=1075.882,49.413,-64.594,173.534,22.993,154.039
C09722=1075.887,49.663,-64.610,173.536,22.996,154.040
C09723=1075.893,49.913,-64.626,173.537,22.999,154.040
C09724=1075.899,50.162,-64.643,173.538,23.001,154.040
C09725=1075.905,50.411,-64.659,173.540,23.003,154.040
C09726=1075.911,50.661,-64.675,173.542,23.006,154.041
C09727=1075.917,50.910,-64.691,173.543,23.009,154.041
C09728=1075.922,51.160,-64.708,173.544,23.011,154.041
C09729=1075.927,51.408,-64.724,173.545,23.014,154.042
C09730=1075.933,51.658,-64.740,173.547,23.017,154.042
C09731=1075.939,51.907,-64.757,173.549,23.019,154.042
C09732=1075.945,52.156,-64.773,173.550,23.022,154.043
C09733=1075.951,52.406,-64.789,173.551,23.024,154.043
C09734=1075.956,52.655,-64.806,173.553,23.027,154.043
C09735=1075.962,52.905,-64.822,173.555,23.029,154.043
C09736=1075.968,53.154,-64.839,173.556,23.032,154.044
C09737=1075.974,53.403,-64.855,173.557,23.034,154.044
C09738=1075.980,53.653,-64.871,173.559,23.037,154.044
C09739=1075.985,53.902,-64.888,173.560,23.039,154.045
C09740=1075.991,54.152,-64.904,173.562,23.042,154.045
C09741=1075.997,54.401,-64.920,173.563,23.044,154.045
C09742=1076.003,54.650,-64.937,173.565,23.047,154.045
C09743=1076.009,54.900,-64.953,173.566,23.049,154.046
C09744=1076.014,55.149,-64.970,173.568,23.052,154.046
C09745=1076.020,55.399,-64.986,173.569,23.055,154.046
C09746=1076.026,55.648,-65.002,173.570,23.057,154.047
C09747=1076.032,55.897,-65.019,173.572,23.060,154.047
C09748=1076.038,56.147,-65.035,173.574,23.063,154.047
C09749=1076.043,56.396,-65.052,173.575,23.065,154.047
C09750=1076.049,56.646,-65.068,173.576,23.067,154.048
C09751=1076.055,56.895,-65.084,173.578,23.070,154.048
C09752=1076.062,57.145,-65.101,173.579,23.072,154.048
C09753=1076.067,57.394,-65.118,173.581,23.075,154.049
C09754=1076.073,57.644,-65.135,173.582,23.077,154.049
C09755=1076.079,57.893,-65.151,173.584,23.080,154.049
C09756=1076.085,58.142,-65.167,173.585,23.082,154.049
C09757=1076.090,58.392,-65.184,173.587,23.085,154.050
C09758=1076.096,58.641,-65.200,173.588,23.087,154.050
C09759=1076.103,58.890,-65.217,173.590,23.090,154.050
C09760=1076.108,59.139,-65.234,173.591,23.092,154.051
C09761=1076.114,59.389,-65.250,173.593,23.095,154.051
C09762=1076.120,59.638,-65.267,173.594,23.097,154.051
C09763=1076.126,59.888,-65.283,173.596,23.100,154.051
C09764=1076.132,60.137,-65.300,173.597,23.102,154.052
C09765=1076.138,60.387,-65.317,173.599,23.105,154.052
C09766=1076.144,60.636,-65.333,173.600,23.107,154.052
C09767=1076.150,60.885,-65.350,173.602,23.110,154.053
C09768=1076.155,61.135,-65.366,173.603,23.112,154.053
C09769=1076.161,61.384,-65.383,173.605,23.115,154.053
C09770=1076.167,61.633,-65.400,173.606,23.118,154.053
C09771=1076.173,61.883,-65.416,173.608,23.120,154.054
C09772=1076.179,62.132,-65.434,173.609,23.122,154.054
C09773=1076.185,62.382,-65.450,173.611,23.125,154.054
C09774=1076.192,62.663,-65.469,173.612,23.128,154.055
C09775=1076.198,62.944,-65.488,173.614,23.130,154.055
C09776=1076.205,63.225,-65.506,173.616,23.133,154.055
C09777=1076.212,63.506,-65.526,173.618,23.136,154.055
C09778=1076.218,63.755,-65.542,173.619,23.139,154.056
C09779=1076.223,64.005,-65.559,173.620,23.141,154.056
C09780=1076.229,64.254,-65.576,173.622,23.143,154.056
C09781=1076.235,64.503,-65.592,173.624,23.146,154.057
C09782=1076.241,64.753,-65.609,173.625,23.149,154.057
C09783=1076.247,65.002,-65.626,173.626,23.151,154.057
C09784=1076.253,65.252,-65.643,173.628,23.153,154.057
C09785=1076.259,65.501,-65.659,173.630,23.156,154.058
C09786=1076.264,65.750,-65.677,173.631,23.159,154.058
C09787=1076.270,65.999,-65.693,173.632,23.161,154.058
C09788=1076.276,66.248,-65.711,173.634,23.163,154.059
C09789=1076.281,66.498,-65.728,173.636,23.166,154.059
C09790=1076.288,66.748,-65.745,173.637,23.169,154.059
C09791=1076.293,66.997,-65.762,173.638,23.171,154.059
C09792=1076.299,67.247,-65.778,173.640,23.173,154.060
C09793=1076.304,67.496,-65.796,173.642,23.176,154.060
C09794=1076.310,67.745,-65.812,173.643,23.179,154.060
C09795=1076.316,67.994,-65.829,173.644,23.181,154.061
C09796=1076.322,68.244,-65.846,173.646,23.183,154.061
C09797=1076.328,68.493,-65.864,173.648,23.186,154.061
C09798=1076.334,68.742,-65.880,173.649,23.189,154.061
C09799=1076.339,68.991,-65.897,173.650,23.191,154.062
C09800=1076.345,69.241,-65.914,173.652,23.194,154.062
C09801=1076.351,69.491,-65.932,173.654,23.196,154.062
C09802=1076.357,69.740,-65.949,173.655,23.199,154.063
C09803=1076.363,69.989,-65.965,173.656,23.201,154.063
C09804=1076.368,70.239,-65.982,173.658,23.204,154.063
C09805=1076.374,70.488,-66.000,173.660,23.206,154.063
C09806=1076.380,70.737,-66.017,173.661,23.209,154.064
C09807=1076.386,70.987,-66.034,173.662,23.212,154.064
C09808=1076.391,71.236,-66.052,173.664,23.214,154.064
C09809=1076.396,71.485,-66.069,173.666,23.217,154.065
C09810=1076.403,71.734,-66.085,173.667,23.219,154.065
C09811=1076.409,71.984,-66.103,173.668,23.222,154.065
C09812=1076.414,72.234,-66.120,173.670,23.224,154.065
C09813=1076.420,72.482,-66.137,173.672,23.227,154.066
C09814=1076.425,72.732,-66.154,173.673,23.229,154.066
C09815=1076.432,72.982,-66.172,173.675,23.232,154.066
C09816=1076.437,73.231,-66.190,173.676,23.234,154.067
C09817=1076.443,73.480,-66.206,173.678,23.237,154.067
C09818=1076.449,73.729,-66.223,173.679,23.239,154.067
C09819=1076.455,73.979,-66.241,173.681,23.242,154.067
C09820=1076.461,74.228,-66.258,173.682,23.244,154.068
C09821=1076.466,74.477,-66.275,173.684,23.247,154.068
C09822=1076.472,74.726,-66.293,173.685,23.249,154.068
C09823=1076.477,74.977,-66.310,173.687,23.252,154.069
C09824=1076.484,75.225,-66.327,173.688,23.254,154.069
C09825=1076.489,75.474,-66.344,173.690,23.257,154.069
C09826=1076.495,75.723,-66.362,173.692,23.260,154.069
C09827=1076.501,75.974,-66.379,173.693,23.262,154.070
C09828=1076.506,76.223,-66.397,173.694,23.264,154.070
C09829=1076.512,76.472,-66.414,173.696,23.267,154.070
C09830=1076.519,76.721,-66.432,173.698,23.270,154.071
C09831=1076.524,76.971,-66.449,173.699,23.272,154.071
C09832=1076.529,77.220,-66.466,173.701,23.274,154.071
C09833=1076.536,77.469,-66.484,173.703,23.277,154.071
C09834=1076.542,77.718,-66.501,173.704,23.280,154.072
C09835=1076.547,77.968,-66.519,173.705,23.282,154.072
C09836=1076.552,78.217,-66.535,173.707,23.284,154.072
C09837=1076.558,78.467,-66.553,173.709,23.287,154.072
C09838=1076.565,78.747,-66.573,173.710,23.290,154.073
C09839=1076.572,79.028,-66.593,173.712,23.292,154.073
C09840=1076.578,79.309,-66.613,173.713,23.295,154.073
C09841=1076.584,79.591,-66.632,173.716,23.298,154.074
C09842=1076.589,79.840,-66.650,173.717,23.300,154.074
C09843=1076.595,80.090,-66.668,173.719,23.303,154.074
C09844=1076.601,80.339,-66.685,173.720,23.306,154.075
C09845=1076.606,80.588,-66.703,173.722,23.308,154.075
C09846=1076.613,80.837,-66.720,173.724,23.311,154.075
C09847=1076.619,81.086,-66.738,173.725,23.313,154.075
C09848=1076.624,81.335,-66.755,173.726,23.316,154.076
C09849=1076.631,81.585,-66.773,173.728,23.318,154.076
C09850=1076.636,81.834,-66.791,173.730,23.321,154.076
C09851=1076.641,82.084,-66.808,173.731,23.323,154.077
C09852=1076.647,82.333,-66.826,173.732,23.326,154.077
C09853=1076.653,82.582,-66.843,173.735,23.328,154.077
C09854=1076.658,82.831,-66.861,173.736,23.331,154.077
C09855=1076.665,83.081,-66.879,173.737,23.333,154.078
C09856=1076.669,83.331,-66.897,173.739,23.336,154.078
C09857=1076.675,83.580,-66.914,173.741,23.338,154.078
C09858=1076.681,83.829,-66.932,173.742,23.341,154.079
C09859=1076.686,84.078,-66.950,173.743,23.343,154.079
C09860=1076.693,84.328,-66.968,173.745,23.346,154.079
C09861=1076.698,84.577,-66.985,173.747,23.348,154.079
C09862=1076.704,84.826,-67.003,173.748,23.351,154.080
C09863=1076.710,85.076,-67.021,173.750,23.354,154.080
C09864=1076.716,85.324,-67.039,173.751,23.356,154.080
C09865=1076.722,85.574,-67.057,173.753,23.358,154.080
C09866=1076.727,85.823,-67.075,173.755,23.361,154.081
C09867=1076.733,86.072,-67.092,173.756,23.363,154.081
C09868=1076.739,86.322,-67.110,173.758,23.366,154.081
C09869=1076.744,86.571,-67.128,173.760,23.369,154.082
C09870=1076.750,86.821,-67.146,173.761,23.371,154.082
C09871=1076.756,87.070,-67.163,173.762,23.373,154.082
C09872=1076.762,87.319,-67.181,173.764,23.376,154.082
C09873=1076.768,87.568,-67.199,173.766,23.379,154.083
C09874=1076.773,87.817,-67.217,173.767,23.380,154.083
C09875=1076.780,88.067,-67.235,173.769,23.383,154.083
C09876=1076.785,88.316,-67.253,173.771,23.386,154.083
C09877=1076.790,88.566,-67.271,173.772,23.388,154.084
C09878=1076.796,88.815,-67.289,173.773,23.390,154.084
C09879=1076.802,89.065,-67.307,173.776,23.393,154.084
C09880=1076.808,89.313,-67.325,173.777,23.396,154.085
C09881=1076.814,89.563,-67.343,173.778,23.398,154.085
C09882=1076.820,89.812,-67.360,173.780,23.401,154.085
C09883=1076.826,90.061,-67.378,173.782,23.403,154.085
C09884=1076.831,90.310,-67.396,173.783,23.405,154.086
C09885=1076.838,90.560,-67.415,173.785,23.408,154.086
C09886=1076.843,90.809,-67.432,173.787,23.410,154.086
C09887=1076.849,91.059,-67.451,173.788,23.413,154.086
C09888=1076.854,91.308,-67.468,173.790,23.415,154.087
C09889=1076.860,91.557,-67.487,173.791,23.418,154.087
C09890=1076.866,91.806,-67.504,173.793,23.420,154.087
C09891=1076.871,92.056,-67.523,173.795,23.423,154.088
C09892=1076.877,92.304,-67.541,173.796,23.425,154.088
C09893=1076.883,92.554,-67.559,173.797,23.428,154.088
C09894=1076.888,92.803,-67.577,173.800,23.430,154.088
C09895=1076.894,93.053,-67.595,173.801,23.433,154.089
C09896=1076.900,93.302,-67.614,173.802,23.435,154.089
C09897=1076.905,93.551,-67.632,173.804,23.438,154.089
C09898=1076.911,93.801,-67.650,173.806,23.440,154.089
C09899=1076.917,94.049,-67.668,173.807,23.443,154.090
C09900=1076.922,94.299,-67.686,173.809,23.445,154.090
C09901=1076.928,94.548,-67.705,173.811,23.447,154.090
C09902=1076.935,94.829,-67.725,173.813,23.451,154.091
C09903=1076.941,95.110,-67.745,173.814,23.453,154.091
C09904=1076.947,95.391,-67.767,173.816,23.456,154.091
C09905=1076.954,95.672,-67.787,173.818,23.459,154.092
C09906=1076.960,95.922,-67.805,173.820,23.461,154.092
C09907=1076.966,96.170,-67.823,173.821,23.463,154.092
C09908=1076.971,96.420,-67.842,173.823,23.466,154.092
C09909=1076.977,96.669,-67.860,173.825,23.469,154.093
C09910=1076.983,96.919,-67.878,173.826,23.471,154.093
C09911=1076.988,97.167,-67.897,173.828,23.474,154.093
C09912=1076.994,97.417,-67.915,173.829,23.476,154.093
C09913=1077.000,97.667,-67.934,173.831,23.479,154.094
C09914=1077.005,97.916,-67.951,173.833,23.481,154.094
C09915=1077.012,98.165,-67.970,173.834,23.483,154.094
C09916=1077.017,98.414,-67.988,173.836,23.486,154.094
C09917=1077.023,98.663,-68.007,173.838,23.488,154.095
C09918=1077.029,98.912,-68.025,173.839,23.491,154.095
C09919=1077.034,99.162,-68.044,173.841,23.493,154.095
C09920=1077.040,99.411,-68.062,173.843,23.496,154.095
C09921=1077.045,99.660,-68.081,173.844,23.498,154.096
C09922=1077.052,99.910,-68.098,173.846,23.500,154.096
C09923=1077.058,100.159,-68.117,173.848,23.503,154.096
C09924=1077.063,100.408,-68.135,173.849,23.505,154.097
C09925=1077.069,100.657,-68.154,173.851,23.508,154.097
C09926=1077.074,100.906,-68.173,173.852,23.510,154.097
C09927=1077.080,101.156,-68.191,173.854,23.512,154.097
C09928=1077.086,101.405,-68.210,173.856,23.515,154.097
C09929=1077.092,101.654,-68.228,173.857,23.517,154.098
C09930=1077.097,101.904,-68.247,173.860,23.520,154.098
C09931=1077.103,102.152,-68.265,173.861,23.523,154.098
C09932=1077.108,102.402,-68.284,173.862,23.525,154.099
C09933=1077.114,102.652,-68.303,173.864,23.528,154.099
C09934=1077.120,102.900,-68.321,173.866,23.530,154.099
C09935=1077.125,103.150,-68.340,173.867,23.532,154.099
C09936=1077.132,103.399,-68.358,173.869,23.535,154.100
C09937=1077.137,103.648,-68.377,173.871,23.537,154.100
C09938=1077.142,103.898,-68.396,173.872,23.539,154.100
C09939=1077.148,104.147,-68.414,173.874,23.542,154.100
C09940=1077.154,104.396,-68.433,173.876,23.545,154.101
C09941=1077.160,104.645,-68.452,173.878,23.547,154.101
C09942=1077.165,104.894,-68.470,173.879,23.550,154.101
C09943=1077.171,105.144,-68.489,173.880,23.552,154.102
C09944=1077.177,105.393,-68.508,173.883,23.555,154.102
C09945=1077.182,105.642,-68.526,173.884,23.557,154.102
C09946=1077.188,105.892,-68.545,173.886,23.560,154.102
C09947=1077.194,106.141,-68.564,173.888,23.562,154.103
C09948=1077.199,106.390,-68.583,173.889,23.564,154.103
C09949=1077.206,106.639,-68.602,173.891,23.567,154.103
C09950=1077.211,106.889,-68.620,173.892,23.569,154.103
C09951=1077.216,107.138,-68.639,173.894,23.571,154.104
C09952=1077.222,107.387,-68.658,173.896,23.574,154.104
C09953=1077.228,107.636,-68.677,173.897,23.576,154.104
C09954=1077.234,107.886,-68.696,173.900,23.579,154.104
C09955=1077.240,108.134,-68.714,173.901,23.582,154.105
C09956=1077.245,108.384,-68.733,173.902,23.583,154.105
C09957=1077.251,108.633,-68.752,173.905,23.586,154.105
C09958=1077.256,108.882,-68.770,173.906,23.589,154.105
C09959=1077.262,109.131,-68.790,173.908,23.591,154.106
C09960=1077.268,109.381,-68.809,173.909,23.594,154.106
C09961=1077.274,109.630,-68.828,173.911,23.596,154.106
C09962=1077.279,109.879,-68.846,173.913,23.598,154.106
C09963=1077.285,110.128,-68.866,173.914,23.601,154.107
C09964=1077.291,110.377,-68.884,173.917,23.603,154.107
C09965=1077.297,110.627,-68.904,173.918,23.605,154.107
C09966=1077.303,110.908,-68.925,173.920,23.609,154.107
C09967=1077.310,111.189,-68.945,173.921,23.611,154.108
C09968=1077.316,111.470,-68.967,173.924,23.614,154.108
C09969=1077.323,111.751,-68.989,173.926,23.616,154.108
C09970=1077.328,112.001,-69.008,173.927,23.619,154.109
C09971=1077.334,112.249,-69.026,173.929,23.622,154.109
C09972=1077.340,112.499,-69.046,173.931,23.623,154.109
C09973=1077.345,112.748,-69.065,173.933,23.626,154.109
C09974=1077.351,112.997,-69.084,173.934,23.629,154.110
C09975=1077.356,113.246,-69.103,173.936,23.631,154.110
C09976=1077.362,113.496,-69.122,173.938,23.634,154.110
C09977=1077.368,113.745,-69.141,173.939,23.636,154.110
C09978=1077.374,113.994,-69.160,173.942,23.638,154.111
C09979=1077.380,114.244,-69.179,173.943,23.641,154.111
C09980=1077.385,114.492,-69.199,173.944,23.643,154.111
C09981=1077.391,114.741,-69.218,173.947,23.645,154.111
C09982=1077.397,114.991,-69.237,173.948,23.648,154.112
C09983=1077.402,115.240,-69.257,173.950,23.650,154.112
C09984=1077.407,115.489,-69.275,173.951,23.653,154.112
C09985=1077.413,115.738,-69.295,173.954,23.656,154.112
C09986=1077.419,115.988,-69.314,173.955,23.658,154.113
C09987=1077.424,116.237,-69.333,173.956,23.660,154.113
C09988=1077.429,116.486,-69.352,173.959,23.663,154.113
C09989=1077.435,116.735,-69.372,173.960,23.665,154.113
C09990=1077.441,116.984,-69.391,173.962,23.668,154.114
C09991=1077.447,117.233,-69.410,173.964,23.670,154.114
C09992=1077.453,117.483,-69.430,173.966,23.673,154.114
C09993=1077.458,117.732,-69.449,173.967,23.675,154.114
C09994=1077.464,117.980,-69.469,173.969,23.677,154.115
C09995=1077.469,118.230,-69.488,173.971,23.680,154.115
C09996=1077.474,118.480,-69.508,173.972,23.682,154.115
//INST
///DATE 2021/06/17 10:54
///ATTR SC,RW,RJ
////FRAME ROBOT
///GROUP1 RB1
NOP
MOVL C00000 V=800.0 PL=0
MOVL C00001 V=800.0 PL=0
MOVL C00002 V=800.0 PL=0
MOVL C00003 V=800.0 PL=0
MOVL C00004 V=800.0 PL=0
MOVL C00005 V=800.0 PL=0
MOVL C00006 V=800.0 PL=0
MOVL C00007 V=800.0 PL=0
MOVL C00008 V=800.0 PL=0
MOVL C00009 V=800.0 PL=0
MOVL C00010 V=800.0 PL=0
MOVL C00011 V=800.0 PL=0
MOVL C00012 V=800.0 PL=0
MOVL C00013 V=800.0 PL=0
MOVL C00014 V=800.0 PL=0
MOVL C00015 V=800.0 PL=0
MOVL C00016 V=800.0 PL=0
MOVL C00017 V=800.0 PL=0
MOVL C00018 V=800.0 PL=0
MOVL C00019 V=800.0 PL=0
MOVL C00020 V=800.0 PL=0
MOVL C00021 V=800.0 PL=0
MOVL C00022 V=800.0 PL=0
MOVL C00023 V=800.0 PL=0
MOVL C00024 V=800.0 PL=0
MOVL C00025 V=800.0 PL=0
MOVL C00026 V=800.0 PL=0
MOVL C00027 V=800.0 PL=0
MOVL C00028 V=800.0 PL=0
MOVL C00029 V=800.0 PL=0
MOVL C00030 V=800.0 PL=0
MOVL C00031 V=800.0 PL=0
MOVL C00032 V=800.0 PL=0
MOVL C00033 V=800.0 PL=0
MOVL C00034 V=800.0 PL=0
MOVL C00035 V=800.0 PL=0
MOVL C00036 V=800.0 PL=0
MOVL C00037 V=800.0 PL=0
MOVL C00038 V=800.0 PL=0
MOVL C00039 V=800.0 PL=0
MOVL C00040 V=800.0 PL=0
MOVL C00041 V=800.0 PL=0
MOVL C00042 V=800.0 PL=0
MOVL C00043 V=800.0 PL=0
MOVL C00044 V=800.0 PL=0
MOVL C00045 V=800.0 PL=0
MOVL C00046 V=800.0 PL=0
MOVL C00047 V=800.0 PL=0
MOVL C00048 V=800.0 PL=0
MOVL C00049 V=800.0 PL=0
MOVL C00050 V=800.0 PL=0
MOVL C00051 V=800.0 PL=0
MOVL C00052 V=800.0 PL=0
MOVL C00053 V=800.0 PL=0
MOVL C00054 V=800.0 PL=0
MOVL C00055 V=800.0 PL=0
MOVL C00056 V=800.0 PL=0
MOVL C00057 V=800.0 PL=0
MOVL C00058 V=800.0 PL=0
MOVL C00059 V=800.0 PL=0
MOVL C00060 V=800.0 PL=0
MOVL C00061 V=800.0 PL=0
MOVL C00062 V=800.0 PL=0
MOVL C00063 V=800.0 PL=0
MOVL C00064 V=800.0 PL=0
MOVL C00065 V=800.0 PL=0
MOVL C00066 V=800.0 PL=0
MOVL C00067 V=800.0 PL=0
MOVL C00068 V=800.0 PL=0
MOVL C00069 V=800.0 PL=0
MOVL C00070 V=800.0 PL=0
MOVL C00071 V=800.0 PL=0
MOVL C00072 V=800.0 PL=0
MOVL C00073 V=800.0 PL=0
MOVL C00074 V=800.0 PL=0
MOVL C00075 V=800.0 PL=0
MOVL C00076 V=800.0 PL=0
MOVL C00077 V=800.0 PL=0
MOVL C00078 V=800.0 PL=0
MOVL C00079 V=800.0 PL=0
MOVL C00080 V=800.0 PL=0
MOVL C00081 V=800.0 PL=0
MOVL C00082 V=800.0 PL=0
MOVL C00083 V=800.0 PL=0
MOVL C00084 V=800.0 PL=0
MOVL C00085 V=800.0 PL=0
MOVL C00086 V=800.0 PL=0
MOVL C00087 V=800.0 PL=0
MOVL C00088 V=800.0 PL=0
MOVL C00089 V=800.0 PL=0
MOVL C00090 V=800.0 PL=0
MOVL C00091 V=800.0 PL=0
MOVL C00092 V=800.0 PL=0
MOVL C00093 V=800.0 PL=0
MOVL C00094 V=800.0 PL=0
MOVL C00095 V=800.0 PL=0
MOVL C00096 V=800.0 PL=0
MOVL C00097 V=800.0 PL=0
MOVL C00098 V=800.0 PL=0
MOVL C00099 V=800.0 PL=0
MOVL C00100 V=800.0 PL=0
MOVL C00101 V=800.0 PL=0
MOVL C00102 V=800.0 PL=0
MOVL C00103 V=800.0 PL=0
MOVL C00104 V=800.0 PL=0
MOVL C00105 V=800.0 PL=0
MOVL C00106 V=800.0 PL=0
MOVL C00107 V=800.0 PL=0
MOVL C00108 V=800.0 PL=0
MOVL C00109 V=800.0 PL=0
MOVL C00110 V=800.0 PL=0
MOVL C00111 V=800.0 PL=0
MOVL C00112 V=800.0 PL=0
MOVL C00113 V=800.0 PL=0
MOVL C00114 V=800.0 PL=0
MOVL C00115 V=800.0 PL=0
MOVL C00116 V=800.0 PL=0
MOVL C00117 V=800.0 PL=0
MOVL C00118 V=800.0 PL=0
MOVL C00119 V=800.0 PL=0
MOVL C00120 V=800.0 PL=0
MOVL C00121 V=800.0 PL=0
MOVL C00122 V=800.0 PL=0
MOVL C00123 V=800.0 PL=0
MOVL C00124 V=800.0 PL=0
MOVL C00125 V=800.0 PL=0
MOVL C00126 V=800.0 PL=0
MOVL C00127 V=800.0 PL=0
MOVL C00128 V=800.0 PL=0
MOVL C00129 V=800.0 PL=0
MOVL C00130 V=800.0 PL=0
MOVL C00131 V=800.0 PL=0
MOVL C00132 V=800.0 PL=0
MOVL C00133 V=800.0 PL=0
MOVL C00134 V=800.0 PL=0
MOVL C00135 V=800.0 PL=0
MOVL C00136 V=800.0 PL=0
MOVL C00137 V=800.0 PL=0
MOVL C00138 V=800.0 PL=0
MOVL C00139 V=800.0 PL=0
MOVL C00140 V=800.0 PL=0
MOVL C00141 V=800.0 PL=0
MOVL C00142 V=800.0 PL=0
MOVL C00143 V=800.0 PL=0
MOVL C00144 V=800.0 PL=0
MOVL C00145 V=800.0 PL=0
MOVL C00146 V=800.0 PL=0
MOVL C00147 V=800.0 PL=0
MOVL C00148 V=800.0 PL=0
MOVL C00149 V=800.0 PL=0
MOVL C00150 V=800.0 PL=0
MOVL C00151 V=800.0 PL=0
MOVL C00152 V=800.0 PL=0
MOVL C00153 V=800.0 PL=0
MOVL C00154 V=800.0 PL=0
MOVL C00155 V=800.0 PL=0
MOVL C00156 V=800.0 PL=0
MOVL C00157 V=800.0 PL=0
MOVL C00158 V=800.0 PL=0
MOVL C00159 V=800.0 PL=0
MOVL C00160 V=800.0 PL=0
MOVL C00161 V=800.0 PL=0
MOVL C00162 V=800.0 PL=0
MOVL C00163 V=800.0 PL=0
MOVL C00164 V=800.0 PL=0
MOVL C00165 V=800.0 PL=0
MOVL C00166 V=800.0 PL=0
MOVL C00167 V=800.0 PL=0
MOVL C00168 V=800.0 PL=0
MOVL C00169 V=800.0 PL=0
MOVL C00170 V=800.0 PL=0
MOVL C00171 V=800.0 PL=0
MOVL C00172 V=800.0 PL=0
MOVL C00173 V=800.0 PL=0
MOVL C00174 V=800.0 PL=0
MOVL C00175 V=800.0 PL=0
MOVL C00176 V=800.0 PL=0
MOVL C00177 V=800.0 PL=0
MOVL C00178 V=800.0 PL=0
MOVL C00179 V=800.0 PL=0
MOVL C00180 V=800.0 PL=0
MOVL C00181 V=800.0 PL=0
MOVL C00182 V=800.0 PL=0
MOVL C00183 V=800.0 PL=0
MOVL C00184 V=800.0 PL=0
MOVL C00185 V=800.0 PL=0
MOVL C00186 V=800.0 PL=0
MOVL C00187 V=800.0 PL=0
MOVL C00188 V=800.0 PL=0
MOVL C00189 V=800.0 PL=0
MOVL C00190 V=800.0 PL=0
MOVL C00191 V=800.0 PL=0
MOVL C00192 V=800.0 PL=0
MOVL C00193 V=800.0 PL=0
MOVL C00194 V=800.0 PL=0
MOVL C00195 V=800.0 PL=0
MOVL C00196 V=800.0 PL=0
MOVL C00197 V=800.0 PL=0
MOVL C00198 V=800.0 PL=0
MOVL C00199 V=800.0 PL=0
MOVL C00200 V=800.0 PL=0
MOVL C00201 V=800.0 PL=0
MOVL C00202 V=800.0 PL=0
MOVL C00203 V=800.0 PL=0
MOVL C00204 V=800.0 PL=0
MOVL C00205 V=800.0 PL=0
MOVL C00206 V=800.0 PL=0
MOVL C00207 V=800.0 PL=0
MOVL C00208 V=800.0 PL=0
MOVL C00209 V=800.0 PL=0
MOVL C00210 V=800.0 PL=0
MOVL C00211 V=800.0 PL=0
MOVL C00212 V=800.0 PL=0
MOVL C00213 V=800.0 PL=0
MOVL C00214 V=800.0 PL=0
MOVL C00215 V=800.0 PL=0
MOVL C00216 V=800.0 PL=0
MOVL C00217 V=800.0 PL=0
MOVL C00218 V=800.0 PL=0
MOVL C00219 V=800.0 PL=0
MOVL C00220 V=800.0 PL=0
MOVL C00221 V=800.0 PL=0
MOVL C00222 V=800.0 PL=0
MOVL C00223 V=800.0 PL=0
MOVL C00224 V=800.0 PL=0
MOVL C00225 V=800.0 PL=0
MOVL C00226 V=800.0 PL=0
MOVL C00227 V=800.0 PL=0
MOVL C00228 V=800.0 PL=0
MOVL C00229 V=800.0 PL=0
MOVL C00230 V=800.0 PL=0
MOVL C00231 V=800.0 PL=0
MOVL C00232 V=800.0 PL=0
MOVL C00233 V=800.0 PL=0
MOVL C00234 V=800.0 PL=0
MOVL C00235 V=800.0 PL=0
MOVL C00236 V=800.0 PL=0
MOVL C00237 V=800.0 PL=0
MOVL C00238 V=800.0 PL=0
MOVL C00239 V=800.0 PL=0
MOVL C00240 V=800.0 PL=0
MOVL C00241 V=800.0 PL=0
MOVL C00242 V=800.0 PL=0
MOVL C00243 V=800.0 PL=0
MOVL C00244 V=800.0 PL=0
MOVL C00245 V=800.0 PL=0
MOVL C00246 V=800.0 PL=0
MOVL C00247 V=800.0 PL=0
MOVL C00248 V=800.0 PL=0
MOVL C00249 V=800.0 PL=0
MOVL C00250 V=800.0 PL=0
MOVL C00251 V=800.0 PL=0
MOVL C00252 V=800.0 PL=0
MOVL C00253 V=800.0 PL=0
MOVL C00254 V=800.0 PL=0
MOVL C00255 V=800.0 PL=0
MOVL C00256 V=800.0 PL=0
MOVL C00257 V=800.0 PL=0
MOVL C00258 V=800.0 PL=0
MOVL C00259 V=800.0 PL=0
MOVL C00260 V=800.0 PL=0
MOVL C00261 V=800.0 PL=0
MOVL C00262 V=800.0 PL=0
MOVL C00263 V=800.0 PL=0
MOVL C00264 V=800.0 PL=0
MOVL C00265 V=800.0 PL=0
MOVL C00266 V=800.0 PL=0
MOVL C00267 V=800.0 PL=0
MOVL C00268 V=800.0 PL=0
MOVL C00269 V=800.0 PL=0
MOVL C00270 V=800.0 PL=0
MOVL C00271 V=800.0 PL=0
MOVL C00272 V=800.0 PL=0
MOVL C00273 V=800.0 PL=0
MOVL C00274 V=800.0 PL=0
MOVL C00275 V=800.0 PL=0
MOVL C00276 V=800.0 PL=0
MOVL C00277 V=800.0 PL=0
MOVL C00278 V=800.0 PL=0
MOVL C00279 V=800.0 PL=0
MOVL C00280 V=800.0 PL=0
MOVL C00281 V=800.0 PL=0
MOVL C00282 V=800.0 PL=0
MOVL C00283 V=800.0 PL=0
MOVL C00284 V=800.0 PL=0
MOVL C00285 V=800.0 PL=0
MOVL C00286 V=800.0 PL=0
MOVL C00287 V=800.0 PL=0
MOVL C00288 V=800.0 PL=0
MOVL C00289 V=800.0 PL=0
MOVL C00290 V=800.0 PL=0
MOVL C00291 V=800.0 PL=0
MOVL C00292 V=800.0 PL=0
MOVL C00293 V=800.0 PL=0
MOVL C00294 V=800.0 PL=0
MOVL C00295 V=800.0 PL=0
MOVL C00296 V=800.0 PL=0
MOVL C00297 V=800.0 PL=0
MOVL C00298 V=800.0 PL=0
MOVL C00299 V=800.0 PL=0
MOVL C00300 V=800.0 PL=0
MOVL C00301 V=800.0 PL=0
MOVL C00302 V=800.0 PL=0
MOVL C00303 V=800.0 PL=0
MOVL C00304 V=800.0 PL=0
MOVL C00305 V=800.0 PL=0
MOVL C00306 V=800.0 PL=0
MOVL C00307 V=800.0 PL=0
MOVL C00308 V=800.0 PL=0
MOVL C00309 V=800.0 PL=0
MOVL C00310 V=800.0 PL=0
MOVL C00311 V=800.0 PL=0
MOVL C00312 V=800.0 PL=0
MOVL C00313 V=800.0 PL=0
MOVL C00314 V=800.0 PL=0
MOVL C00315 V=800.0 PL=0
MOVL C00316 V=800.0 PL=0
MOVL C00317 V=800.0 PL=0
MOVL C00318 V=800.0 PL=0
MOVL C00319 V=800.0 PL=0
MOVL C00320 V=800.0 PL=0
MOVL C00321 V=800.0 PL=0
MOVL C00322 V=800.0 PL=0
MOVL C00323 V=800.0 PL=0
MOVL C00324 V=800.0 PL=0
MOVL C00325 V=800.0 PL=0
MOVL C00326 V=800.0 PL=0
MOVL C00327 V=800.0 PL=0
MOVL C00328 V=800.0 PL=0
MOVL C00329 V=800.0 PL=0
MOVL C00330 V=800.0 PL=0
MOVL C00331 V=800.0 PL=0
MOVL C00332 V=800.0 PL=0
MOVL C00333 V=800.0 PL=0
MOVL C00334 V=800.0 PL=0
MOVL C00335 V=800.0 PL=0
MOVL C00336 V=800.0 PL=0
MOVL C00337 V=800.0 PL=0
MOVL C00338 V=800.0 PL=0
MOVL C00339 V=800.0 PL=0
MOVL C00340 V=800.0 PL=0
MOVL C00341 V=800.0 PL=0
MOVL C00342 V=800.0 PL=0
MOVL C00343 V=800.0 PL=0
MOVL C00344 V=800.0 PL=0
MOVL C00345 V=800.0 PL=0
MOVL C00346 V=800.0 PL=0
MOVL C00347 V=800.0 PL=0
MOVL C00348 V=800.0 PL=0
MOVL C00349 V=800.0 PL=0
MOVL C00350 V=800.0 PL=0
MOVL C00351 V=800.0 PL=0
MOVL C00352 V=800.0 PL=0
MOVL C00353 V=800.0 PL=0
MOVL C00354 V=800.0 PL=0
MOVL C00355 V=800.0 PL=0
MOVL C00356 V=800.0 PL=0
MOVL C00357 V=800.0 PL=0
MOVL C00358 V=800.0 PL=0
MOVL C00359 V=800.0 PL=0
MOVL C00360 V=800.0 PL=0
MOVL C00361 V=800.0 PL=0
MOVL C00362 V=800.0 PL=0
MOVL C00363 V=800.0 PL=0
MOVL C00364 V=800.0 PL=0
MOVL C00365 V=800.0 PL=0
MOVL C00366 V=800.0 PL=0
MOVL C00367 V=800.0 PL=0
MOVL C00368 V=800.0 PL=0
MOVL C00369 V=800.0 PL=0
MOVL C00370 V=800.0 PL=0
MOVL C00371 V=800.0 PL=0
MOVL C00372 V=800.0 PL=0
MOVL C00373 V=800.0 PL=0
MOVL C00374 V=800.0 PL=0
MOVL C00375 V=800.0 PL=0
MOVL C00376 V=800.0 PL=0
MOVL C00377 V=800.0 PL=0
MOVL C00378 V=800.0 PL=0
MOVL C00379 V=800.0 PL=0
MOVL C00380 V=800.0 PL=0
MOVL C00381 V=800.0 PL=0
MOVL C00382 V=800.0 PL=0
MOVL C00383 V=800.0 PL=0
MOVL C00384 V=800.0 PL=0
MOVL C00385 V=800.0 PL=0
MOVL C00386 V=800.0 PL=0
MOVL C00387 V=800.0 PL=0
MOVL C00388 V=800.0 PL=0
MOVL C00389 V=800.0 PL=0
MOVL C00390 V=800.0 PL=0
MOVL C00391 V=800.0 PL=0
MOVL C00392 V=800.0 PL=0
MOVL C00393 V=800.0 PL=0
MOVL C00394 V=800.0 PL=0
MOVL C00395 V=800.0 PL=0
MOVL C00396 V=800.0 PL=0
MOVL C00397 V=800.0 PL=0
MOVL C00398 V=800.0 PL=0
MOVL C00399 V=800.0 PL=0
MOVL C00400 V=800.0 PL=0
MOVL C00401 V=800.0 PL=0
MOVL C00402 V=800.0 PL=0
MOVL C00403 V=800.0 PL=0
MOVL C00404 V=800.0 PL=0
MOVL C00405 V=800.0 PL=0
MOVL C00406 V=800.0 PL=0
MOVL C00407 V=800.0 PL=0
MOVL C00408 V=800.0 PL=0
MOVL C00409 V=800.0 PL=0
MOVL C00410 V=800.0 PL=0
MOVL C00411 V=800.0 PL=0
MOVL C00412 V=800.0 PL=0
MOVL C00413 V=800.0 PL=0
MOVL C00414 V=800.0 PL=0
MOVL C00415 V=800.0 PL=0
MOVL C00416 V=800.0 PL=0
MOVL C00417 V=800.0 PL=0
MOVL C00418 V=800.0 PL=0
MOVL C00419 V=800.0 PL=0
MOVL C00420 V=800.0 PL=0
MOVL C00421 V=800.0 PL=0
MOVL C00422 V=800.0 PL=0
MOVL C00423 V=800.0 PL=0
MOVL C00424 V=800.0 PL=0
MOVL C00425 V=800.0 PL=0
MOVL C00426 V=800.0 PL=0
MOVL C00427 V=800.0 PL=0
MOVL C00428 V=800.0 PL=0
MOVL C00429 V=800.0 PL=0
MOVL C00430 V=800.0 PL=0
MOVL C00431 V=800.0 PL=0
MOVL C00432 V=800.0 PL=0
MOVL C00433 V=800.0 PL=0
MOVL C00434 V=800.0 PL=0
MOVL C00435 V=800.0 PL=0
MOVL C00436 V=800.0 PL=0
MOVL C00437 V=800.0 PL=0
MOVL C00438 V=800.0 PL=0
MOVL C00439 V=800.0 PL=0
MOVL C00440 V=800.0 PL=0
MOVL C00441 V=800.0 PL=0
MOVL C00442 V=800.0 PL=0
MOVL C00443 V=800.0 PL=0
MOVL C00444 V=800.0 PL=0
MOVL C00445 V=800.0 PL=0
MOVL C00446 V=800.0 PL=0
MOVL C00447 V=800.0 PL=0
MOVL C00448 V=800.0 PL=0
MOVL C00449 V=800.0 PL=0
MOVL C00450 V=800.0 PL=0
MOVL C00451 V=800.0 PL=0
MOVL C00452 V=800.0 PL=0
MOVL C00453 V=800.0 PL=0
MOVL C00454 V=800.0 PL=0
MOVL C00455 V=800.0 PL=0
MOVL C00456 V=800.0 PL=0
MOVL C00457 V=800.0 PL=0
MOVL C00458 V=800.0 PL=0
MOVL C00459 V=800.0 PL=0
MOVL C00460 V=800.0 PL=0
MOVL C00461 V=800.0 PL=0
MOVL C00462 V=800.0 PL=0
MOVL C00463 V=800.0 PL=0
MOVL C00464 V=800.0 PL=0
MOVL C00465 V=800.0 PL=0
MOVL C00466 V=800.0 PL=0
MOVL C00467 V=800.0 PL=0
MOVL C00468 V=800.0 PL=0
MOVL C00469 V=800.0 PL=0
MOVL C00470 V=800.0 PL=0
MOVL C00471 V=800.0 PL=0
MOVL C00472 V=800.0 PL=0
MOVL C00473 V=800.0 PL=0
MOVL C00474 V=800.0 PL=0
MOVL C00475 V=800.0 PL=0
MOVL C00476 V=800.0 PL=0
MOVL C00477 V=800.0 PL=0
MOVL C00478 V=800.0 PL=0
MOVL C00479 V=800.0 PL=0
MOVL C00480 V=800.0 PL=0
MOVL C00481 V=800.0 PL=0
MOVL C00482 V=800.0 PL=0
MOVL C00483 V=800.0 PL=0
MOVL C00484 V=800.0 PL=0
MOVL C00485 V=800.0 PL=0
MOVL C00486 V=800.0 PL=0
MOVL C00487 V=800.0 PL=0
MOVL C00488 V=800.0 PL=0
MOVL C00489 V=800.0 PL=0
MOVL C00490 V=800.0 PL=0
MOVL C00491 V=800.0 PL=0
MOVL C00492 V=800.0 PL=0
MOVL C00493 V=800.0 PL=0
MOVL C00494 V=800.0 PL=0
MOVL C00495 V=800.0 PL=0
MOVL C00496 V=800.0 PL=0
MOVL C00497 V=800.0 PL=0
MOVL C00498 V=800.0 PL=0
MOVL C00499 V=800.0 PL=0
MOVL C00500 V=800.0 PL=0
MOVL C00501 V=800.0 PL=0
MOVL C00502 V=800.0 PL=0
MOVL C00503 V=800.0 PL=0
MOVL C00504 V=800.0 PL=0
MOVL C00505 V=800.0 PL=0
MOVL C00506 V=800.0 PL=0
MOVL C00507 V=800.0 PL=0
MOVL C00508 V=800.0 PL=0
MOVL C00509 V=800.0 PL=0
MOVL C00510 V=800.0 PL=0
MOVL C00511 V=800.0 PL=0
MOVL C00512 V=800.0 PL=0
MOVL C00513 V=800.0 PL=0
MOVL C00514 V=800.0 PL=0
MOVL C00515 V=800.0 PL=0
MOVL C00516 V=800.0 PL=0
MOVL C00517 V=800.0 PL=0
MOVL C00518 V=800.0 PL=0
MOVL C00519 V=800.0 PL=0
MOVL C00520 V=800.0 PL=0
MOVL C00521 V=800.0 PL=0
MOVL C00522 V=800.0 PL=0
MOVL C00523 V=800.0 PL=0
MOVL C00524 V=800.0 PL=0
MOVL C00525 V=800.0 PL=0
MOVL C00526 V=800.0 PL=0
MOVL C00527 V=800.0 PL=0
MOVL C00528 V=800.0 PL=0
MOVL C00529 V=800.0 PL=0
MOVL C00530 V=800.0 PL=0
MOVL C00531 V=800.0 PL=0
MOVL C00532 V=800.0 PL=0
MOVL C00533 V=800.0 PL=0
MOVL C00534 V=800.0 PL=0
MOVL C00535 V=800.0 PL=0
MOVL C00536 V=800.0 PL=0
MOVL C00537 V=800.0 PL=0
MOVL C00538 V=800.0 PL=0
MOVL C00539 V=800.0 PL=0
MOVL C00540 V=800.0 PL=0
MOVL C00541 V=800.0 PL=0
MOVL C00542 V=800.0 PL=0
MOVL C00543 V=800.0 PL=0
MOVL C00544 V=800.0 PL=0
MOVL C00545 V=800.0 PL=0
MOVL C00546 V=800.0 PL=0
MOVL C00547 V=800.0 PL=0
MOVL C00548 V=800.0 PL=0
MOVL C00549 V=800.0 PL=0
MOVL C00550 V=800.0 PL=0
MOVL C00551 V=800.0 PL=0
MOVL C00552 V=800.0 PL=0
MOVL C00553 V=800.0 PL=0
MOVL C00554 V=800.0 PL=0
MOVL C00555 V=800.0 PL=0
MOVL C00556 V=800.0 PL=0
MOVL C00557 V=800.0 PL=0
MOVL C00558 V=800.0 PL=0
MOVL C00559 V=800.0 PL=0
MOVL C00560 V=800.0 PL=0
MOVL C00561 V=800.0 PL=0
MOVL C00562 V=800.0 PL=0
MOVL C00563 V=800.0 PL=0
MOVL C00564 V=800.0 PL=0
MOVL C00565 V=800.0 PL=0
MOVL C00566 V=800.0 PL=0
MOVL C00567 V=800.0 PL=0
MOVL C00568 V=800.0 PL=0
MOVL C00569 V=800.0 PL=0
MOVL C00570 V=800.0 PL=0
MOVL C00571 V=800.0 PL=0
MOVL C00572 V=800.0 PL=0
MOVL C00573 V=800.0 PL=0
MOVL C00574 V=800.0 PL=0
MOVL C00575 V=800.0 PL=0
MOVL C00576 V=800.0 PL=0
MOVL C00577 V=800.0 PL=0
MOVL C00578 V=800.0 PL=0
MOVL C00579 V=800.0 PL=0
MOVL C00580 V=800.0 PL=0
MOVL C00581 V=800.0 PL=0
MOVL C00582 V=800.0 PL=0
MOVL C00583 V=800.0 PL=0
MOVL C00584 V=800.0 PL=0
MOVL C00585 V=800.0 PL=0
MOVL C00586 V=800.0 PL=0
MOVL C00587 V=800.0 PL=0
MOVL C00588 V=800.0 PL=0
MOVL C00589 V=800.0 PL=0
MOVL C00590 V=800.0 PL=0
MOVL C00591 V=800.0 PL=0
MOVL C00592 V=800.0 PL=0
MOVL C00593 V=800.0 PL=0
MOVL C00594 V=800.0 PL=0
MOVL C00595 V=800.0 PL=0
MOVL C00596 V=800.0 PL=0
MOVL C00597 V=800.0 PL=0
MOVL C00598 V=800.0 PL=0
MOVL C00599 V=800.0 PL=0
MOVL C00600 V=800.0 PL=0
MOVL C00601 V=800.0 PL=0
MOVL C00602 V=800.0 PL=0
MOVL C00603 V=800.0 PL=0
MOVL C00604 V=800.0 PL=0
MOVL C00605 V=800.0 PL=0
MOVL C00606 V=800.0 PL=0
MOVL C00607 V=800.0 PL=0
MOVL C00608 V=800.0 PL=0
MOVL C00609 V=800.0 PL=0
MOVL C00610 V=800.0 PL=0
MOVL C00611 V=800.0 PL=0
MOVL C00612 V=800.0 PL=0
MOVL C00613 V=800.0 PL=0
MOVL C00614 V=800.0 PL=0
MOVL C00615 V=800.0 PL=0
MOVL C00616 V=800.0 PL=0
MOVL C00617 V=800.0 PL=0
MOVL C00618 V=800.0 PL=0
MOVL C00619 V=800.0 PL=0
MOVL C00620 V=800.0 PL=0
MOVL C00621 V=800.0 PL=0
MOVL C00622 V=800.0 PL=0
MOVL C00623 V=800.0 PL=0
MOVL C00624 V=800.0 PL=0
MOVL C00625 V=800.0 PL=0
MOVL C00626 V=800.0 PL=0
MOVL C00627 V=800.0 PL=0
MOVL C00628 V=800.0 PL=0
MOVL C00629 V=800.0 PL=0
MOVL C00630 V=800.0 PL=0
MOVL C00631 V=800.0 PL=0
MOVL C00632 V=800.0 PL=0
MOVL C00633 V=800.0 PL=0
MOVL C00634 V=800.0 PL=0
MOVL C00635 V=800.0 PL=0
MOVL C00636 V=800.0 PL=0
MOVL C00637 V=800.0 PL=0
MOVL C00638 V=800.0 PL=0
MOVL C00639 V=800.0 PL=0
MOVL C00640 V=800.0 PL=0
MOVL C00641 V=800.0 PL=0
MOVL C00642 V=800.0 PL=0
MOVL C00643 V=800.0 PL=0
MOVL C00644 V=800.0 PL=0
MOVL C00645 V=800.0 PL=0
MOVL C00646 V=800.0 PL=0
MOVL C00647 V=800.0 PL=0
MOVL C00648 V=800.0 PL=0
MOVL C00649 V=800.0 PL=0
MOVL C00650 V=800.0 PL=0
MOVL C00651 V=800.0 PL=0
MOVL C00652 V=800.0 PL=0
MOVL C00653 V=800.0 PL=0
MOVL C00654 V=800.0 PL=0
MOVL C00655 V=800.0 PL=0
MOVL C00656 V=800.0 PL=0
MOVL C00657 V=800.0 PL=0
MOVL C00658 V=800.0 PL=0
MOVL C00659 V=800.0 PL=0
MOVL C00660 V=800.0 PL=0
MOVL C00661 V=800.0 PL=0
MOVL C00662 V=800.0 PL=0
MOVL C00663 V=800.0 PL=0
MOVL C00664 V=800.0 PL=0
MOVL C00665 V=800.0 PL=0
MOVL C00666 V=800.0 PL=0
MOVL C00667 V=800.0 PL=0
MOVL C00668 V=800.0 PL=0
MOVL C00669 V=800.0 PL=0
MOVL C00670 V=800.0 PL=0
MOVL C00671 V=800.0 PL=0
MOVL C00672 V=800.0 PL=0
MOVL C00673 V=800.0 PL=0
MOVL C00674 V=800.0 PL=0
MOVL C00675 V=800.0 PL=0
MOVL C00676 V=800.0 PL=0
MOVL C00677 V=800.0 PL=0
MOVL C00678 V=800.0 PL=0
MOVL C00679 V=800.0 PL=0
MOVL C00680 V=800.0 PL=0
MOVL C00681 V=800.0 PL=0
MOVL C00682 V=800.0 PL=0
MOVL C00683 V=800.0 PL=0
MOVL C00684 V=800.0 PL=0
MOVL C00685 V=800.0 PL=0
MOVL C00686 V=800.0 PL=0
MOVL C00687 V=800.0 PL=0
MOVL C00688 V=800.0 PL=0
MOVL C00689 V=800.0 PL=0
MOVL C00690 V=800.0 PL=0
MOVL C00691 V=800.0 PL=0
MOVL C00692 V=800.0 PL=0
MOVL C00693 V=800.0 PL=0
MOVL C00694 V=800.0 PL=0
MOVL C00695 V=800.0 PL=0
MOVL C00696 V=800.0 PL=0
MOVL C00697 V=800.0 PL=0
MOVL C00698 V=800.0 PL=0
MOVL C00699 V=800.0 PL=0
MOVL C00700 V=800.0 PL=0
MOVL C00701 V=800.0 PL=0
MOVL C00702 V=800.0 PL=0
MOVL C00703 V=800.0 PL=0
MOVL C00704 V=800.0 PL=0
MOVL C00705 V=800.0 PL=0
MOVL C00706 V=800.0 PL=0
MOVL C00707 V=800.0 PL=0
MOVL C00708 V=800.0 PL=0
MOVL C00709 V=800.0 PL=0
MOVL C00710 V=800.0 PL=0
MOVL C00711 V=800.0 PL=0
MOVL C00712 V=800.0 PL=0
MOVL C00713 V=800.0 PL=0
MOVL C00714 V=800.0 PL=0
MOVL C00715 V=800.0 PL=0
MOVL C00716 V=800.0 PL=0
MOVL C00717 V=800.0 PL=0
MOVL C00718 V=800.0 PL=0
MOVL C00719 V=800.0 PL=0
MOVL C00720 V=800.0 PL=0
MOVL C00721 V=800.0 PL=0
MOVL C00722 V=800.0 PL=0
MOVL C00723 V=800.0 PL=0
MOVL C00724 V=800.0 PL=0
MOVL C00725 V=800.0 PL=0
MOVL C00726 V=800.0 PL=0
MOVL C00727 V=800.0 PL=0
MOVL C00728 V=800.0 PL=0
MOVL C00729 V=800.0 PL=0
MOVL C00730 V=800.0 PL=0
MOVL C00731 V=800.0 PL=0
MOVL C00732 V=800.0 PL=0
MOVL C00733 V=800.0 PL=0
MOVL C00734 V=800.0 PL=0
MOVL C00735 V=800.0 PL=0
MOVL C00736 V=800.0 PL=0
MOVL C00737 V=800.0 PL=0
MOVL C00738 V=800.0 PL=0
MOVL C00739 V=800.0 PL=0
MOVL C00740 V=800.0 PL=0
MOVL C00741 V=800.0 PL=0
MOVL C00742 V=800.0 PL=0
MOVL C00743 V=800.0 PL=0
MOVL C00744 V=800.0 PL=0
MOVL C00745 V=800.0 PL=0
MOVL C00746 V=800.0 PL=0
MOVL C00747 V=800.0 PL=0
MOVL C00748 V=800.0 PL=0
MOVL C00749 V=800.0 PL=0
MOVL C00750 V=800.0 PL=0
MOVL C00751 V=800.0 PL=0
MOVL C00752 V=800.0 PL=0
MOVL C00753 V=800.0 PL=0
MOVL C00754 V=800.0 PL=0
MOVL C00755 V=800.0 PL=0
MOVL C00756 V=800.0 PL=0
MOVL C00757 V=800.0 PL=0
MOVL C00758 V=800.0 PL=0
MOVL C00759 V=800.0 PL=0
MOVL C00760 V=800.0 PL=0
MOVL C00761 V=800.0 PL=0
MOVL C00762 V=800.0 PL=0
MOVL C00763 V=800.0 PL=0
MOVL C00764 V=800.0 PL=0
MOVL C00765 V=800.0 PL=0
MOVL C00766 V=800.0 PL=0
MOVL C00767 V=800.0 PL=0
MOVL C00768 V=800.0 PL=0
MOVL C00769 V=800.0 PL=0
MOVL C00770 V=800.0 PL=0
MOVL C00771 V=800.0 PL=0
MOVL C00772 V=800.0 PL=0
MOVL C00773 V=800.0 PL=0
MOVL C00774 V=800.0 PL=0
MOVL C00775 V=800.0 PL=0
MOVL C00776 V=800.0 PL=0
MOVL C00777 V=800.0 PL=0
MOVL C00778 V=800.0 PL=0
MOVL C00779 V=800.0 PL=0
MOVL C00780 V=800.0 PL=0
MOVL C00781 V=800.0 PL=0
MOVL C00782 V=800.0 PL=0
MOVL C00783 V=800.0 PL=0
MOVL C00784 V=800.0 PL=0
MOVL C00785 V=800.0 PL=0
MOVL C00786 V=800.0 PL=0
MOVL C00787 V=800.0 PL=0
MOVL C00788 V=800.0 PL=0
MOVL C00789 V=800.0 PL=0
MOVL C00790 V=800.0 PL=0
MOVL C00791 V=800.0 PL=0
MOVL C00792 V=800.0 PL=0
MOVL C00793 V=800.0 PL=0
MOVL C00794 V=800.0 PL=0
MOVL C00795 V=800.0 PL=0
MOVL C00796 V=800.0 PL=0
MOVL C00797 V=800.0 PL=0
MOVL C00798 V=800.0 PL=0
MOVL C00799 V=800.0 PL=0
MOVL C00800 V=800.0 PL=0
MOVL C00801 V=800.0 PL=0
MOVL C00802 V=800.0 PL=0
MOVL C00803 V=800.0 PL=0
MOVL C00804 V=800.0 PL=0
MOVL C00805 V=800.0 PL=0
MOVL C00806 V=800.0 PL=0
MOVL C00807 V=800.0 PL=0
MOVL C00808 V=800.0 PL=0
MOVL C00809 V=800.0 PL=0
MOVL C00810 V=800.0 PL=0
MOVL C00811 V=800.0 PL=0
MOVL C00812 V=800.0 PL=0
MOVL C00813 V=800.0 PL=0
MOVL C00814 V=800.0 PL=0
MOVL C00815 V=800.0 PL=0
MOVL C00816 V=800.0 PL=0
MOVL C00817 V=800.0 PL=0
MOVL C00818 V=800.0 PL=0
MOVL C00819 V=800.0 PL=0
MOVL C00820 V=800.0 PL=0
MOVL C00821 V=800.0 PL=0
MOVL C00822 V=800.0 PL=0
MOVL C00823 V=800.0 PL=0
MOVL C00824 V=800.0 PL=0
MOVL C00825 V=800.0 PL=0
MOVL C00826 V=800.0 PL=0
MOVL C00827 V=800.0 PL=0
MOVL C00828 V=800.0 PL=0
MOVL C00829 V=800.0 PL=0
MOVL C00830 V=800.0 PL=0
MOVL C00831 V=800.0 PL=0
MOVL C00832 V=800.0 PL=0
MOVL C00833 V=800.0 PL=0
MOVL C00834 V=800.0 PL=0
MOVL C00835 V=800.0 PL=0
MOVL C00836 V=800.0 PL=0
MOVL C00837 V=800.0 PL=0
MOVL C00838 V=800.0 PL=0
MOVL C00839 V=800.0 PL=0
MOVL C00840 V=800.0 PL=0
MOVL C00841 V=800.0 PL=0
MOVL C00842 V=800.0 PL=0
MOVL C00843 V=800.0 PL=0
MOVL C00844 V=800.0 PL=0
MOVL C00845 V=800.0 PL=0
MOVL C00846 V=800.0 PL=0
MOVL C00847 V=800.0 PL=0
MOVL C00848 V=800.0 PL=0
MOVL C00849 V=800.0 PL=0
MOVL C00850 V=800.0 PL=0
MOVL C00851 V=800.0 PL=0
MOVL C00852 V=800.0 PL=0
MOVL C00853 V=800.0 PL=0
MOVL C00854 V=800.0 PL=0
MOVL C00855 V=800.0 PL=0
MOVL C00856 V=800.0 PL=0
MOVL C00857 V=800.0 PL=0
MOVL C00858 V=800.0 PL=0
MOVL C00859 V=800.0 PL=0
MOVL C00860 V=800.0 PL=0
MOVL C00861 V=800.0 PL=0
MOVL C00862 V=800.0 PL=0
MOVL C00863 V=800.0 PL=0
MOVL C00864 V=800.0 PL=0
MOVL C00865 V=800.0 PL=0
MOVL C00866 V=800.0 PL=0
MOVL C00867 V=800.0 PL=0
MOVL C00868 V=800.0 PL=0
MOVL C00869 V=800.0 PL=0
MOVL C00870 V=800.0 PL=0
MOVL C00871 V=800.0 PL=0
MOVL C00872 V=800.0 PL=0
MOVL C00873 V=800.0 PL=0
MOVL C00874 V=800.0 PL=0
MOVL C00875 V=800.0 PL=0
MOVL C00876 V=800.0 PL=0
MOVL C00877 V=800.0 PL=0
MOVL C00878 V=800.0 PL=0
MOVL C00879 V=800.0 PL=0
MOVL C00880 V=800.0 PL=0
MOVL C00881 V=800.0 PL=0
MOVL C00882 V=800.0 PL=0
MOVL C00883 V=800.0 PL=0
MOVL C00884 V=800.0 PL=0
MOVL C00885 V=800.0 PL=0
MOVL C00886 V=800.0 PL=0
MOVL C00887 V=800.0 PL=0
MOVL C00888 V=800.0 PL=0
MOVL C00889 V=800.0 PL=0
MOVL C00890 V=800.0 PL=0
MOVL C00891 V=800.0 PL=0
MOVL C00892 V=800.0 PL=0
MOVL C00893 V=800.0 PL=0
MOVL C00894 V=800.0 PL=0
MOVL C00895 V=800.0 PL=0
MOVL C00896 V=800.0 PL=0
MOVL C00897 V=800.0 PL=0
MOVL C00898 V=800.0 PL=0
MOVL C00899 V=800.0 PL=0
MOVL C00900 V=800.0 PL=0
MOVL C00901 V=800.0 PL=0
MOVL C00902 V=800.0 PL=0
MOVL C00903 V=800.0 PL=0
MOVL C00904 V=800.0 PL=0
MOVL C00905 V=800.0 PL=0
MOVL C00906 V=800.0 PL=0
MOVL C00907 V=800.0 PL=0
MOVL C00908 V=800.0 PL=0
MOVL C00909 V=800.0 PL=0
MOVL C00910 V=800.0 PL=0
MOVL C00911 V=800.0 PL=0
MOVL C00912 V=800.0 PL=0
MOVL C00913 V=800.0 PL=0
MOVL C00914 V=800.0 PL=0
MOVL C00915 V=800.0 PL=0
MOVL C00916 V=800.0 PL=0
MOVL C00917 V=800.0 PL=0
MOVL C00918 V=800.0 PL=0
MOVL C00919 V=800.0 PL=0
MOVL C00920 V=800.0 PL=0
MOVL C00921 V=800.0 PL=0
MOVL C00922 V=800.0 PL=0
MOVL C00923 V=800.0 PL=0
MOVL C00924 V=800.0 PL=0
MOVL C00925 V=800.0 PL=0
MOVL C00926 V=800.0 PL=0
MOVL C00927 V=800.0 PL=0
MOVL C00928 V=800.0 PL=0
MOVL C00929 V=800.0 PL=0
MOVL C00930 V=800.0 PL=0
MOVL C00931 V=800.0 PL=0
MOVL C00932 V=800.0 PL=0
MOVL C00933 V=800.0 PL=0
MOVL C00934 V=800.0 PL=0
MOVL C00935 V=800.0 PL=0
MOVL C00936 V=800.0 PL=0
MOVL C00937 V=800.0 PL=0
MOVL C00938 V=800.0 PL=0
MOVL C00939 V=800.0 PL=0
MOVL C00940 V=800.0 PL=0
MOVL C00941 V=800.0 PL=0
MOVL C00942 V=800.0 PL=0
MOVL C00943 V=800.0 PL=0
MOVL C00944 V=800.0 PL=0
MOVL C00945 V=800.0 PL=0
MOVL C00946 V=800.0 PL=0
MOVL C00947 V=800.0 PL=0
MOVL C00948 V=800.0 PL=0
MOVL C00949 V=800.0 PL=0
MOVL C00950 V=800.0 PL=0
MOVL C00951 V=800.0 PL=0
MOVL C00952 V=800.0 PL=0
MOVL C00953 V=800.0 PL=0
MOVL C00954 V=800.0 PL=0
MOVL C00955 V=800.0 PL=0
MOVL C00956 V=800.0 PL=0
MOVL C00957 V=800.0 PL=0
MOVL C00958 V=800.0 PL=0
MOVL C00959 V=800.0 PL=0
MOVL C00960 V=800.0 PL=0
MOVL C00961 V=800.0 PL=0
MOVL C00962 V=800.0 PL=0
MOVL C00963 V=800.0 PL=0
MOVL C00964 V=800.0 PL=0
MOVL C00965 V=800.0 PL=0
MOVL C00966 V=800.0 PL=0
MOVL C00967 V=800.0 PL=0
MOVL C00968 V=800.0 PL=0
MOVL C00969 V=800.0 PL=0
MOVL C00970 V=800.0 PL=0
MOVL C00971 V=800.0 PL=0
MOVL C00972 V=800.0 PL=0
MOVL C00973 V=800.0 PL=0
MOVL C00974 V=800.0 PL=0
MOVL C00975 V=800.0 PL=0
MOVL C00976 V=800.0 PL=0
MOVL C00977 V=800.0 PL=0
MOVL C00978 V=800.0 PL=0
MOVL C00979 V=800.0 PL=0
MOVL C00980 V=800.0 PL=0
MOVL C00981 V=800.0 PL=0
MOVL C00982 V=800.0 PL=0
MOVL C00983 V=800.0 PL=0
MOVL C00984 V=800.0 PL=0
MOVL C00985 V=800.0 PL=0
MOVL C00986 V=800.0 PL=0
MOVL C00987 V=800.0 PL=0
MOVL C00988 V=800.0 PL=0
MOVL C00989 V=800.0 PL=0
MOVL C00990 V=800.0 PL=0
MOVL C00991 V=800.0 PL=0
MOVL C00992 V=800.0 PL=0
MOVL C00993 V=800.0 PL=0
MOVL C00994 V=800.0 PL=0
MOVL C00995 V=800.0 PL=0
MOVL C00996 V=800.0 PL=0
MOVL C00997 V=800.0 PL=0
MOVL C00998 V=800.0 PL=0
MOVL C00999 V=800.0 PL=0
MOVL C01000 V=800.0 PL=0
MOVL C01001 V=800.0 PL=0
MOVL C01002 V=800.0 PL=0
MOVL C01003 V=800.0 PL=0
MOVL C01004 V=800.0 PL=0
MOVL C01005 V=800.0 PL=0
MOVL C01006 V=800.0 PL=0
MOVL C01007 V=800.0 PL=0
MOVL C01008 V=800.0 PL=0
MOVL C01009 V=800.0 PL=0
MOVL C01010 V=800.0 PL=0
MOVL C01011 V=800.0 PL=0
MOVL C01012 V=800.0 PL=0
MOVL C01013 V=800.0 PL=0
MOVL C01014 V=800.0 PL=0
MOVL C01015 V=800.0 PL=0
MOVL C01016 V=800.0 PL=0
MOVL C01017 V=800.0 PL=0
MOVL C01018 V=800.0 PL=0
MOVL C01019 V=800.0 PL=0
MOVL C01020 V=800.0 PL=0
MOVL C01021 V=800.0 PL=0
MOVL C01022 V=800.0 PL=0
MOVL C01023 V=800.0 PL=0
MOVL C01024 V=800.0 PL=0
MOVL C01025 V=800.0 PL=0
MOVL C01026 V=800.0 PL=0
MOVL C01027 V=800.0 PL=0
MOVL C01028 V=800.0 PL=0
MOVL C01029 V=800.0 PL=0
MOVL C01030 V=800.0 PL=0
MOVL C01031 V=800.0 PL=0
MOVL C01032 V=800.0 PL=0
MOVL C01033 V=800.0 PL=0
MOVL C01034 V=800.0 PL=0
MOVL C01035 V=800.0 PL=0
MOVL C01036 V=800.0 PL=0
MOVL C01037 V=800.0 PL=0
MOVL C01038 V=800.0 PL=0
MOVL C01039 V=800.0 PL=0
MOVL C01040 V=800.0 PL=0
MOVL C01041 V=800.0 PL=0
MOVL C01042 V=800.0 PL=0
MOVL C01043 V=800.0 PL=0
MOVL C01044 V=800.0 PL=0
MOVL C01045 V=800.0 PL=0
MOVL C01046 V=800.0 PL=0
MOVL C01047 V=800.0 PL=0
MOVL C01048 V=800.0 PL=0
MOVL C01049 V=800.0 PL=0
MOVL C01050 V=800.0 PL=0
MOVL C01051 V=800.0 PL=0
MOVL C01052 V=800.0 PL=0
MOVL C01053 V=800.0 PL=0
MOVL C01054 V=800.0 PL=0
MOVL C01055 V=800.0 PL=0
MOVL C01056 V=800.0 PL=0
MOVL C01057 V=800.0 PL=0
MOVL C01058 V=800.0 PL=0
MOVL C01059 V=800.0 PL=0
MOVL C01060 V=800.0 PL=0
MOVL C01061 V=800.0 PL=0
MOVL C01062 V=800.0 PL=0
MOVL C01063 V=800.0 PL=0
MOVL C01064 V=800.0 PL=0
MOVL C01065 V=800.0 PL=0
MOVL C01066 V=800.0 PL=0
MOVL C01067 V=800.0 PL=0
MOVL C01068 V=800.0 PL=0
MOVL C01069 V=800.0 PL=0
MOVL C01070 V=800.0 PL=0
MOVL C01071 V=800.0 PL=0
MOVL C01072 V=800.0 PL=0
MOVL C01073 V=800.0 PL=0
MOVL C01074 V=800.0 PL=0
MOVL C01075 V=800.0 PL=0
MOVL C01076 V=800.0 PL=0
MOVL C01077 V=800.0 PL=0
MOVL C01078 V=800.0 PL=0
MOVL C01079 V=800.0 PL=0
MOVL C01080 V=800.0 PL=0
MOVL C01081 V=800.0 PL=0
MOVL C01082 V=800.0 PL=0
MOVL C01083 V=800.0 PL=0
MOVL C01084 V=800.0 PL=0
MOVL C01085 V=800.0 PL=0
MOVL C01086 V=800.0 PL=0
MOVL C01087 V=800.0 PL=0
MOVL C01088 V=800.0 PL=0
MOVL C01089 V=800.0 PL=0
MOVL C01090 V=800.0 PL=0
MOVL C01091 V=800.0 PL=0
MOVL C01092 V=800.0 PL=0
MOVL C01093 V=800.0 PL=0
MOVL C01094 V=800.0 PL=0
MOVL C01095 V=800.0 PL=0
MOVL C01096 V=800.0 PL=0
MOVL C01097 V=800.0 PL=0
MOVL C01098 V=800.0 PL=0
MOVL C01099 V=800.0 PL=0
MOVL C01100 V=800.0 PL=0
MOVL C01101 V=800.0 PL=0
MOVL C01102 V=800.0 PL=0
MOVL C01103 V=800.0 PL=0
MOVL C01104 V=800.0 PL=0
MOVL C01105 V=800.0 PL=0
MOVL C01106 V=800.0 PL=0
MOVL C01107 V=800.0 PL=0
MOVL C01108 V=800.0 PL=0
MOVL C01109 V=800.0 PL=0
MOVL C01110 V=800.0 PL=0
MOVL C01111 V=800.0 PL=0
MOVL C01112 V=800.0 PL=0
MOVL C01113 V=800.0 PL=0
MOVL C01114 V=800.0 PL=0
MOVL C01115 V=800.0 PL=0
MOVL C01116 V=800.0 PL=0
MOVL C01117 V=800.0 PL=0
MOVL C01118 V=800.0 PL=0
MOVL C01119 V=800.0 PL=0
MOVL C01120 V=800.0 PL=0
MOVL C01121 V=800.0 PL=0
MOVL C01122 V=800.0 PL=0
MOVL C01123 V=800.0 PL=0
MOVL C01124 V=800.0 PL=0
MOVL C01125 V=800.0 PL=0
MOVL C01126 V=800.0 PL=0
MOVL C01127 V=800.0 PL=0
MOVL C01128 V=800.0 PL=0
MOVL C01129 V=800.0 PL=0
MOVL C01130 V=800.0 PL=0
MOVL C01131 V=800.0 PL=0
MOVL C01132 V=800.0 PL=0
MOVL C01133 V=800.0 PL=0
MOVL C01134 V=800.0 PL=0
MOVL C01135 V=800.0 PL=0
MOVL C01136 V=800.0 PL=0
MOVL C01137 V=800.0 PL=0
MOVL C01138 V=800.0 PL=0
MOVL C01139 V=800.0 PL=0
MOVL C01140 V=800.0 PL=0
MOVL C01141 V=800.0 PL=0
MOVL C01142 V=800.0 PL=0
MOVL C01143 V=800.0 PL=0
MOVL C01144 V=800.0 PL=0
MOVL C01145 V=800.0 PL=0
MOVL C01146 V=800.0 PL=0
MOVL C01147 V=800.0 PL=0
MOVL C01148 V=800.0 PL=0
MOVL C01149 V=800.0 PL=0
MOVL C01150 V=800.0 PL=0
MOVL C01151 V=800.0 PL=0
MOVL C01152 V=800.0 PL=0
MOVL C01153 V=800.0 PL=0
MOVL C01154 V=800.0 PL=0
MOVL C01155 V=800.0 PL=0
MOVL C01156 V=800.0 PL=0
MOVL C01157 V=800.0 PL=0
MOVL C01158 V=800.0 PL=0
MOVL C01159 V=800.0 PL=0
MOVL C01160 V=800.0 PL=0
MOVL C01161 V=800.0 PL=0
MOVL C01162 V=800.0 PL=0
MOVL C01163 V=800.0 PL=0
MOVL C01164 V=800.0 PL=0
MOVL C01165 V=800.0 PL=0
MOVL C01166 V=800.0 PL=0
MOVL C01167 V=800.0 PL=0
MOVL C01168 V=800.0 PL=0
MOVL C01169 V=800.0 PL=0
MOVL C01170 V=800.0 PL=0
MOVL C01171 V=800.0 PL=0
MOVL C01172 V=800.0 PL=0
MOVL C01173 V=800.0 PL=0
MOVL C01174 V=800.0 PL=0
MOVL C01175 V=800.0 PL=0
MOVL C01176 V=800.0 PL=0
MOVL C01177 V=800.0 PL=0
MOVL C01178 V=800.0 PL=0
MOVL C01179 V=800.0 PL=0
MOVL C01180 V=800.0 PL=0
MOVL C01181 V=800.0 PL=0
MOVL C01182 V=800.0 PL=0
MOVL C01183 V=800.0 PL=0
MOVL C01184 V=800.0 PL=0
MOVL C01185 V=800.0 PL=0
MOVL C01186 V=800.0 PL=0
MOVL C01187 V=800.0 PL=0
MOVL C01188 V=800.0 PL=0
MOVL C01189 V=800.0 PL=0
MOVL C01190 V=800.0 PL=0
MOVL C01191 V=800.0 PL=0
MOVL C01192 V=800.0 PL=0
MOVL C01193 V=800.0 PL=0
MOVL C01194 V=800.0 PL=0
MOVL C01195 V=800.0 PL=0
MOVL C01196 V=800.0 PL=0
MOVL C01197 V=800.0 PL=0
MOVL C01198 V=800.0 PL=0
MOVL C01199 V=800.0 PL=0
MOVL C01200 V=800.0 PL=0
MOVL C01201 V=800.0 PL=0
MOVL C01202 V=800.0 PL=0
MOVL C01203 V=800.0 PL=0
MOVL C01204 V=800.0 PL=0
MOVL C01205 V=800.0 PL=0
MOVL C01206 V=800.0 PL=0
MOVL C01207 V=800.0 PL=0
MOVL C01208 V=800.0 PL=0
MOVL C01209 V=800.0 PL=0
MOVL C01210 V=800.0 PL=0
MOVL C01211 V=800.0 PL=0
MOVL C01212 V=800.0 PL=0
MOVL C01213 V=800.0 PL=0
MOVL C01214 V=800.0 PL=0
MOVL C01215 V=800.0 PL=0
MOVL C01216 V=800.0 PL=0
MOVL C01217 V=800.0 PL=0
MOVL C01218 V=800.0 PL=0
MOVL C01219 V=800.0 PL=0
MOVL C01220 V=800.0 PL=0
MOVL C01221 V=800.0 PL=0
MOVL C01222 V=800.0 PL=0
MOVL C01223 V=800.0 PL=0
MOVL C01224 V=800.0 PL=0
MOVL C01225 V=800.0 PL=0
MOVL C01226 V=800.0 PL=0
MOVL C01227 V=800.0 PL=0
MOVL C01228 V=800.0 PL=0
MOVL C01229 V=800.0 PL=0
MOVL C01230 V=800.0 PL=0
MOVL C01231 V=800.0 PL=0
MOVL C01232 V=800.0 PL=0
MOVL C01233 V=800.0 PL=0
MOVL C01234 V=800.0 PL=0
MOVL C01235 V=800.0 PL=0
MOVL C01236 V=800.0 PL=0
MOVL C01237 V=800.0 PL=0
MOVL C01238 V=800.0 PL=0
MOVL C01239 V=800.0 PL=0
MOVL C01240 V=800.0 PL=0
MOVL C01241 V=800.0 PL=0
MOVL C01242 V=800.0 PL=0
MOVL C01243 V=800.0 PL=0
MOVL C01244 V=800.0 PL=0
MOVL C01245 V=800.0 PL=0
MOVL C01246 V=800.0 PL=0
MOVL C01247 V=800.0 PL=0
MOVL C01248 V=800.0 PL=0
MOVL C01249 V=800.0 PL=0
MOVL C01250 V=800.0 PL=0
MOVL C01251 V=800.0 PL=0
MOVL C01252 V=800.0 PL=0
MOVL C01253 V=800.0 PL=0
MOVL C01254 V=800.0 PL=0
MOVL C01255 V=800.0 PL=0
MOVL C01256 V=800.0 PL=0
MOVL C01257 V=800.0 PL=0
MOVL C01258 V=800.0 PL=0
MOVL C01259 V=800.0 PL=0
MOVL C01260 V=800.0 PL=0
MOVL C01261 V=800.0 PL=0
MOVL C01262 V=800.0 PL=0
MOVL C01263 V=800.0 PL=0
MOVL C01264 V=800.0 PL=0
MOVL C01265 V=800.0 PL=0
MOVL C01266 V=800.0 PL=0
MOVL C01267 V=800.0 PL=0
MOVL C01268 V=800.0 PL=0
MOVL C01269 V=800.0 PL=0
MOVL C01270 V=800.0 PL=0
MOVL C01271 V=800.0 PL=0
MOVL C01272 V=800.0 PL=0
MOVL C01273 V=800.0 PL=0
MOVL C01274 V=800.0 PL=0
MOVL C01275 V=800.0 PL=0
MOVL C01276 V=800.0 PL=0
MOVL C01277 V=800.0 PL=0
MOVL C01278 V=800.0 PL=0
MOVL C01279 V=800.0 PL=0
MOVL C01280 V=800.0 PL=0
MOVL C01281 V=800.0 PL=0
MOVL C01282 V=800.0 PL=0
MOVL C01283 V=800.0 PL=0
MOVL C01284 V=800.0 PL=0
MOVL C01285 V=800.0 PL=0
MOVL C01286 V=800.0 PL=0
MOVL C01287 V=800.0 PL=0
MOVL C01288 V=800.0 PL=0
MOVL C01289 V=800.0 PL=0
MOVL C01290 V=800.0 PL=0
MOVL C01291 V=800.0 PL=0
MOVL C01292 V=800.0 PL=0
MOVL C01293 V=800.0 PL=0
MOVL C01294 V=800.0 PL=0
MOVL C01295 V=800.0 PL=0
MOVL C01296 V=800.0 PL=0
MOVL C01297 V=800.0 PL=0
MOVL C01298 V=800.0 PL=0
MOVL C01299 V=800.0 PL=0
MOVL C01300 V=800.0 PL=0
MOVL C01301 V=800.0 PL=0
MOVL C01302 V=800.0 PL=0
MOVL C01303 V=800.0 PL=0
MOVL C01304 V=800.0 PL=0
MOVL C01305 V=800.0 PL=0
MOVL C01306 V=800.0 PL=0
MOVL C01307 V=800.0 PL=0
MOVL C01308 V=800.0 PL=0
MOVL C01309 V=800.0 PL=0
MOVL C01310 V=800.0 PL=0
MOVL C01311 V=800.0 PL=0
MOVL C01312 V=800.0 PL=0
MOVL C01313 V=800.0 PL=0
MOVL C01314 V=800.0 PL=0
MOVL C01315 V=800.0 PL=0
MOVL C01316 V=800.0 PL=0
MOVL C01317 V=800.0 PL=0
MOVL C01318 V=800.0 PL=0
MOVL C01319 V=800.0 PL=0
MOVL C01320 V=800.0 PL=0
MOVL C01321 V=800.0 PL=0
MOVL C01322 V=800.0 PL=0
MOVL C01323 V=800.0 PL=0
MOVL C01324 V=800.0 PL=0
MOVL C01325 V=800.0 PL=0
MOVL C01326 V=800.0 PL=0
MOVL C01327 V=800.0 PL=0
MOVL C01328 V=800.0 PL=0
MOVL C01329 V=800.0 PL=0
MOVL C01330 V=800.0 PL=0
MOVL C01331 V=800.0 PL=0
MOVL C01332 V=800.0 PL=0
MOVL C01333 V=800.0 PL=0
MOVL C01334 V=800.0 PL=0
MOVL C01335 V=800.0 PL=0
MOVL C01336 V=800.0 PL=0
MOVL C01337 V=800.0 PL=0
MOVL C01338 V=800.0 PL=0
MOVL C01339 V=800.0 PL=0
MOVL C01340 V=800.0 PL=0
MOVL C01341 V=800.0 PL=0
MOVL C01342 V=800.0 PL=0
MOVL C01343 V=800.0 PL=0
MOVL C01344 V=800.0 PL=0
MOVL C01345 V=800.0 PL=0
MOVL C01346 V=800.0 PL=0
MOVL C01347 V=800.0 PL=0
MOVL C01348 V=800.0 PL=0
MOVL C01349 V=800.0 PL=0
MOVL C01350 V=800.0 PL=0
MOVL C01351 V=800.0 PL=0
MOVL C01352 V=800.0 PL=0
MOVL C01353 V=800.0 PL=0
MOVL C01354 V=800.0 PL=0
MOVL C01355 V=800.0 PL=0
MOVL C01356 V=800.0 PL=0
MOVL C01357 V=800.0 PL=0
MOVL C01358 V=800.0 PL=0
MOVL C01359 V=800.0 PL=0
MOVL C01360 V=800.0 PL=0
MOVL C01361 V=800.0 PL=0
MOVL C01362 V=800.0 PL=0
MOVL C01363 V=800.0 PL=0
MOVL C01364 V=800.0 PL=0
MOVL C01365 V=800.0 PL=0
MOVL C01366 V=800.0 PL=0
MOVL C01367 V=800.0 PL=0
MOVL C01368 V=800.0 PL=0
MOVL C01369 V=800.0 PL=0
MOVL C01370 V=800.0 PL=0
MOVL C01371 V=800.0 PL=0
MOVL C01372 V=800.0 PL=0
MOVL C01373 V=800.0 PL=0
MOVL C01374 V=800.0 PL=0
MOVL C01375 V=800.0 PL=0
MOVL C01376 V=800.0 PL=0
MOVL C01377 V=800.0 PL=0
MOVL C01378 V=800.0 PL=0
MOVL C01379 V=800.0 PL=0
MOVL C01380 V=800.0 PL=0
MOVL C01381 V=800.0 PL=0
MOVL C01382 V=800.0 PL=0
MOVL C01383 V=800.0 PL=0
MOVL C01384 V=800.0 PL=0
MOVL C01385 V=800.0 PL=0
MOVL C01386 V=800.0 PL=0
MOVL C01387 V=800.0 PL=0
MOVL C01388 V=800.0 PL=0
MOVL C01389 V=800.0 PL=0
MOVL C01390 V=800.0 PL=0
MOVL C01391 V=800.0 PL=0
MOVL C01392 V=800.0 PL=0
MOVL C01393 V=800.0 PL=0
MOVL C01394 V=800.0 PL=0
MOVL C01395 V=800.0 PL=0
MOVL C01396 V=800.0 PL=0
MOVL C01397 V=800.0 PL=0
MOVL C01398 V=800.0 PL=0
MOVL C01399 V=800.0 PL=0
MOVL C01400 V=800.0 PL=0
MOVL C01401 V=800.0 PL=0
MOVL C01402 V=800.0 PL=0
MOVL C01403 V=800.0 PL=0
MOVL C01404 V=800.0 PL=0
MOVL C01405 V=800.0 PL=0
MOVL C01406 V=800.0 PL=0
MOVL C01407 V=800.0 PL=0
MOVL C01408 V=800.0 PL=0
MOVL C01409 V=800.0 PL=0
MOVL C01410 V=800.0 PL=0
MOVL C01411 V=800.0 PL=0
MOVL C01412 V=800.0 PL=0
MOVL C01413 V=800.0 PL=0
MOVL C01414 V=800.0 PL=0
MOVL C01415 V=800.0 PL=0
MOVL C01416 V=800.0 PL=0
MOVL C01417 V=800.0 PL=0
MOVL C01418 V=800.0 PL=0
MOVL C01419 V=800.0 PL=0
MOVL C01420 V=800.0 PL=0
MOVL C01421 V=800.0 PL=0
MOVL C01422 V=800.0 PL=0
MOVL C01423 V=800.0 PL=0
MOVL C01424 V=800.0 PL=0
MOVL C01425 V=800.0 PL=0
MOVL C01426 V=800.0 PL=0
MOVL C01427 V=800.0 PL=0
MOVL C01428 V=800.0 PL=0
MOVL C01429 V=800.0 PL=0
MOVL C01430 V=800.0 PL=0
MOVL C01431 V=800.0 PL=0
MOVL C01432 V=800.0 PL=0
MOVL C01433 V=800.0 PL=0
MOVL C01434 V=800.0 PL=0
MOVL C01435 V=800.0 PL=0
MOVL C01436 V=800.0 PL=0
MOVL C01437 V=800.0 PL=0
MOVL C01438 V=800.0 PL=0
MOVL C01439 V=800.0 PL=0
MOVL C01440 V=800.0 PL=0
MOVL C01441 V=800.0 PL=0
MOVL C01442 V=800.0 PL=0
MOVL C01443 V=800.0 PL=0
MOVL C01444 V=800.0 PL=0
MOVL C01445 V=800.0 PL=0
MOVL C01446 V=800.0 PL=0
MOVL C01447 V=800.0 PL=0
MOVL C01448 V=800.0 PL=0
MOVL C01449 V=800.0 PL=0
MOVL C01450 V=800.0 PL=0
MOVL C01451 V=800.0 PL=0
MOVL C01452 V=800.0 PL=0
MOVL C01453 V=800.0 PL=0
MOVL C01454 V=800.0 PL=0
MOVL C01455 V=800.0 PL=0
MOVL C01456 V=800.0 PL=0
MOVL C01457 V=800.0 PL=0
MOVL C01458 V=800.0 PL=0
MOVL C01459 V=800.0 PL=0
MOVL C01460 V=800.0 PL=0
MOVL C01461 V=800.0 PL=0
MOVL C01462 V=800.0 PL=0
MOVL C01463 V=800.0 PL=0
MOVL C01464 V=800.0 PL=0
MOVL C01465 V=800.0 PL=0
MOVL C01466 V=800.0 PL=0
MOVL C01467 V=800.0 PL=0
MOVL C01468 V=800.0 PL=0
MOVL C01469 V=800.0 PL=0
MOVL C01470 V=800.0 PL=0
MOVL C01471 V=800.0 PL=0
MOVL C01472 V=800.0 PL=0
MOVL C01473 V=800.0 PL=0
MOVL C01474 V=800.0 PL=0
MOVL C01475 V=800.0 PL=0
MOVL C01476 V=800.0 PL=0
MOVL C01477 V=800.0 PL=0
MOVL C01478 V=800.0 PL=0
MOVL C01479 V=800.0 PL=0
MOVL C01480 V=800.0 PL=0
MOVL C01481 V=800.0 PL=0
MOVL C01482 V=800.0 PL=0
MOVL C01483 V=800.0 PL=0
MOVL C01484 V=800.0 PL=0
MOVL C01485 V=800.0 PL=0
MOVL C01486 V=800.0 PL=0
MOVL C01487 V=800.0 PL=0
MOVL C01488 V=800.0 PL=0
MOVL C01489 V=800.0 PL=0
MOVL C01490 V=800.0 PL=0
MOVL C01491 V=800.0 PL=0
MOVL C01492 V=800.0 PL=0
MOVL C01493 V=800.0 PL=0
MOVL C01494 V=800.0 PL=0
MOVL C01495 V=800.0 PL=0
MOVL C01496 V=800.0 PL=0
MOVL C01497 V=800.0 PL=0
MOVL C01498 V=800.0 PL=0
MOVL C01499 V=800.0 PL=0
MOVL C01500 V=800.0 PL=0
MOVL C01501 V=800.0 PL=0
MOVL C01502 V=800.0 PL=0
MOVL C01503 V=800.0 PL=0
MOVL C01504 V=800.0 PL=0
MOVL C01505 V=800.0 PL=0
MOVL C01506 V=800.0 PL=0
MOVL C01507 V=800.0 PL=0
MOVL C01508 V=800.0 PL=0
MOVL C01509 V=800.0 PL=0
MOVL C01510 V=800.0 PL=0
MOVL C01511 V=800.0 PL=0
MOVL C01512 V=800.0 PL=0
MOVL C01513 V=800.0 PL=0
MOVL C01514 V=800.0 PL=0
MOVL C01515 V=800.0 PL=0
MOVL C01516 V=800.0 PL=0
MOVL C01517 V=800.0 PL=0
MOVL C01518 V=800.0 PL=0
MOVL C01519 V=800.0 PL=0
MOVL C01520 V=800.0 PL=0
MOVL C01521 V=800.0 PL=0
MOVL C01522 V=800.0 PL=0
MOVL C01523 V=800.0 PL=0
MOVL C01524 V=800.0 PL=0
MOVL C01525 V=800.0 PL=0
MOVL C01526 V=800.0 PL=0
MOVL C01527 V=800.0 PL=0
MOVL C01528 V=800.0 PL=0
MOVL C01529 V=800.0 PL=0
MOVL C01530 V=800.0 PL=0
MOVL C01531 V=800.0 PL=0
MOVL C01532 V=800.0 PL=0
MOVL C01533 V=800.0 PL=0
MOVL C01534 V=800.0 PL=0
MOVL C01535 V=800.0 PL=0
MOVL C01536 V=800.0 PL=0
MOVL C01537 V=800.0 PL=0
MOVL C01538 V=800.0 PL=0
MOVL C01539 V=800.0 PL=0
MOVL C01540 V=800.0 PL=0
MOVL C01541 V=800.0 PL=0
MOVL C01542 V=800.0 PL=0
MOVL C01543 V=800.0 PL=0
MOVL C01544 V=800.0 PL=0
MOVL C01545 V=800.0 PL=0
MOVL C01546 V=800.0 PL=0
MOVL C01547 V=800.0 PL=0
MOVL C01548 V=800.0 PL=0
MOVL C01549 V=800.0 PL=0
MOVL C01550 V=800.0 PL=0
MOVL C01551 V=800.0 PL=0
MOVL C01552 V=800.0 PL=0
MOVL C01553 V=800.0 PL=0
MOVL C01554 V=800.0 PL=0
MOVL C01555 V=800.0 PL=0
MOVL C01556 V=800.0 PL=0
MOVL C01557 V=800.0 PL=0
MOVL C01558 V=800.0 PL=0
MOVL C01559 V=800.0 PL=0
MOVL C01560 V=800.0 PL=0
MOVL C01561 V=800.0 PL=0
MOVL C01562 V=800.0 PL=0
MOVL C01563 V=800.0 PL=0
MOVL C01564 V=800.0 PL=0
MOVL C01565 V=800.0 PL=0
MOVL C01566 V=800.0 PL=0
MOVL C01567 V=800.0 PL=0
MOVL C01568 V=800.0 PL=0
MOVL C01569 V=800.0 PL=0
MOVL C01570 V=800.0 PL=0
MOVL C01571 V=800.0 PL=0
MOVL C01572 V=800.0 PL=0
MOVL C01573 V=800.0 PL=0
MOVL C01574 V=800.0 PL=0
MOVL C01575 V=800.0 PL=0
MOVL C01576 V=800.0 PL=0
MOVL C01577 V=800.0 PL=0
MOVL C01578 V=800.0 PL=0
MOVL C01579 V=800.0 PL=0
MOVL C01580 V=800.0 PL=0
MOVL C01581 V=800.0 PL=0
MOVL C01582 V=800.0 PL=0
MOVL C01583 V=800.0 PL=0
MOVL C01584 V=800.0 PL=0
MOVL C01585 V=800.0 PL=0
MOVL C01586 V=800.0 PL=0
MOVL C01587 V=800.0 PL=0
MOVL C01588 V=800.0 PL=0
MOVL C01589 V=800.0 PL=0
MOVL C01590 V=800.0 PL=0
MOVL C01591 V=800.0 PL=0
MOVL C01592 V=800.0 PL=0
MOVL C01593 V=800.0 PL=0
MOVL C01594 V=800.0 PL=0
MOVL C01595 V=800.0 PL=0
MOVL C01596 V=800.0 PL=0
MOVL C01597 V=800.0 PL=0
MOVL C01598 V=800.0 PL=0
MOVL C01599 V=800.0 PL=0
MOVL C01600 V=800.0 PL=0
MOVL C01601 V=800.0 PL=0
MOVL C01602 V=800.0 PL=0
MOVL C01603 V=800.0 PL=0
MOVL C01604 V=800.0 PL=0
MOVL C01605 V=800.0 PL=0
MOVL C01606 V=800.0 PL=0
MOVL C01607 V=800.0 PL=0
MOVL C01608 V=800.0 PL=0
MOVL C01609 V=800.0 PL=0
MOVL C01610 V=800.0 PL=0
MOVL C01611 V=800.0 PL=0
MOVL C01612 V=800.0 PL=0
MOVL C01613 V=800.0 PL=0
MOVL C01614 V=800.0 PL=0
MOVL C01615 V=800.0 PL=0
MOVL C01616 V=800.0 PL=0
MOVL C01617 V=800.0 PL=0
MOVL C01618 V=800.0 PL=0
MOVL C01619 V=800.0 PL=0
MOVL C01620 V=800.0 PL=0
MOVL C01621 V=800.0 PL=0
MOVL C01622 V=800.0 PL=0
MOVL C01623 V=800.0 PL=0
MOVL C01624 V=800.0 PL=0
MOVL C01625 V=800.0 PL=0
MOVL C01626 V=800.0 PL=0
MOVL C01627 V=800.0 PL=0
MOVL C01628 V=800.0 PL=0
MOVL C01629 V=800.0 PL=0
MOVL C01630 V=800.0 PL=0
MOVL C01631 V=800.0 PL=0
MOVL C01632 V=800.0 PL=0
MOVL C01633 V=800.0 PL=0
MOVL C01634 V=800.0 PL=0
MOVL C01635 V=800.0 PL=0
MOVL C01636 V=800.0 PL=0
MOVL C01637 V=800.0 PL=0
MOVL C01638 V=800.0 PL=0
MOVL C01639 V=800.0 PL=0
MOVL C01640 V=800.0 PL=0
MOVL C01641 V=800.0 PL=0
MOVL C01642 V=800.0 PL=0
MOVL C01643 V=800.0 PL=0
MOVL C01644 V=800.0 PL=0
MOVL C01645 V=800.0 PL=0
MOVL C01646 V=800.0 PL=0
MOVL C01647 V=800.0 PL=0
MOVL C01648 V=800.0 PL=0
MOVL C01649 V=800.0 PL=0
MOVL C01650 V=800.0 PL=0
MOVL C01651 V=800.0 PL=0
MOVL C01652 V=800.0 PL=0
MOVL C01653 V=800.0 PL=0
MOVL C01654 V=800.0 PL=0
MOVL C01655 V=800.0 PL=0
MOVL C01656 V=800.0 PL=0
MOVL C01657 V=800.0 PL=0
MOVL C01658 V=800.0 PL=0
MOVL C01659 V=800.0 PL=0
MOVL C01660 V=800.0 PL=0
MOVL C01661 V=800.0 PL=0
MOVL C01662 V=800.0 PL=0
MOVL C01663 V=800.0 PL=0
MOVL C01664 V=800.0 PL=0
MOVL C01665 V=800.0 PL=0
MOVL C01666 V=800.0 PL=0
MOVL C01667 V=800.0 PL=0
MOVL C01668 V=800.0 PL=0
MOVL C01669 V=800.0 PL=0
MOVL C01670 V=800.0 PL=0
MOVL C01671 V=800.0 PL=0
MOVL C01672 V=800.0 PL=0
MOVL C01673 V=800.0 PL=0
MOVL C01674 V=800.0 PL=0
MOVL C01675 V=800.0 PL=0
MOVL C01676 V=800.0 PL=0
MOVL C01677 V=800.0 PL=0
MOVL C01678 V=800.0 PL=0
MOVL C01679 V=800.0 PL=0
MOVL C01680 V=800.0 PL=0
MOVL C01681 V=800.0 PL=0
MOVL C01682 V=800.0 PL=0
MOVL C01683 V=800.0 PL=0
MOVL C01684 V=800.0 PL=0
MOVL C01685 V=800.0 PL=0
MOVL C01686 V=800.0 PL=0
MOVL C01687 V=800.0 PL=0
MOVL C01688 V=800.0 PL=0
MOVL C01689 V=800.0 PL=0
MOVL C01690 V=800.0 PL=0
MOVL C01691 V=800.0 PL=0
MOVL C01692 V=800.0 PL=0
MOVL C01693 V=800.0 PL=0
MOVL C01694 V=800.0 PL=0
MOVL C01695 V=800.0 PL=0
MOVL C01696 V=800.0 PL=0
MOVL C01697 V=800.0 PL=0
MOVL C01698 V=800.0 PL=0
MOVL C01699 V=800.0 PL=0
MOVL C01700 V=800.0 PL=0
MOVL C01701 V=800.0 PL=0
MOVL C01702 V=800.0 PL=0
MOVL C01703 V=800.0 PL=0
MOVL C01704 V=800.0 PL=0
MOVL C01705 V=800.0 PL=0
MOVL C01706 V=800.0 PL=0
MOVL C01707 V=800.0 PL=0
MOVL C01708 V=800.0 PL=0
MOVL C01709 V=800.0 PL=0
MOVL C01710 V=800.0 PL=0
MOVL C01711 V=800.0 PL=0
MOVL C01712 V=800.0 PL=0
MOVL C01713 V=800.0 PL=0
MOVL C01714 V=800.0 PL=0
MOVL C01715 V=800.0 PL=0
MOVL C01716 V=800.0 PL=0
MOVL C01717 V=800.0 PL=0
MOVL C01718 V=800.0 PL=0
MOVL C01719 V=800.0 PL=0
MOVL C01720 V=800.0 PL=0
MOVL C01721 V=800.0 PL=0
MOVL C01722 V=800.0 PL=0
MOVL C01723 V=800.0 PL=0
MOVL C01724 V=800.0 PL=0
MOVL C01725 V=800.0 PL=0
MOVL C01726 V=800.0 PL=0
MOVL C01727 V=800.0 PL=0
MOVL C01728 V=800.0 PL=0
MOVL C01729 V=800.0 PL=0
MOVL C01730 V=800.0 PL=0
MOVL C01731 V=800.0 PL=0
MOVL C01732 V=800.0 PL=0
MOVL C01733 V=800.0 PL=0
MOVL C01734 V=800.0 PL=0
MOVL C01735 V=800.0 PL=0
MOVL C01736 V=800.0 PL=0
MOVL C01737 V=800.0 PL=0
MOVL C01738 V=800.0 PL=0
MOVL C01739 V=800.0 PL=0
MOVL C01740 V=800.0 PL=0
MOVL C01741 V=800.0 PL=0
MOVL C01742 V=800.0 PL=0
MOVL C01743 V=800.0 PL=0
MOVL C01744 V=800.0 PL=0
MOVL C01745 V=800.0 PL=0
MOVL C01746 V=800.0 PL=0
MOVL C01747 V=800.0 PL=0
MOVL C01748 V=800.0 PL=0
MOVL C01749 V=800.0 PL=0
MOVL C01750 V=800.0 PL=0
MOVL C01751 V=800.0 PL=0
MOVL C01752 V=800.0 PL=0
MOVL C01753 V=800.0 PL=0
MOVL C01754 V=800.0 PL=0
MOVL C01755 V=800.0 PL=0
MOVL C01756 V=800.0 PL=0
MOVL C01757 V=800.0 PL=0
MOVL C01758 V=800.0 PL=0
MOVL C01759 V=800.0 PL=0
MOVL C01760 V=800.0 PL=0
MOVL C01761 V=800.0 PL=0
MOVL C01762 V=800.0 PL=0
MOVL C01763 V=800.0 PL=0
MOVL C01764 V=800.0 PL=0
MOVL C01765 V=800.0 PL=0
MOVL C01766 V=800.0 PL=0
MOVL C01767 V=800.0 PL=0
MOVL C01768 V=800.0 PL=0
MOVL C01769 V=800.0 PL=0
MOVL C01770 V=800.0 PL=0
MOVL C01771 V=800.0 PL=0
MOVL C01772 V=800.0 PL=0
MOVL C01773 V=800.0 PL=0
MOVL C01774 V=800.0 PL=0
MOVL C01775 V=800.0 PL=0
MOVL C01776 V=800.0 PL=0
MOVL C01777 V=800.0 PL=0
MOVL C01778 V=800.0 PL=0
MOVL C01779 V=800.0 PL=0
MOVL C01780 V=800.0 PL=0
MOVL C01781 V=800.0 PL=0
MOVL C01782 V=800.0 PL=0
MOVL C01783 V=800.0 PL=0
MOVL C01784 V=800.0 PL=0
MOVL C01785 V=800.0 PL=0
MOVL C01786 V=800.0 PL=0
MOVL C01787 V=800.0 PL=0
MOVL C01788 V=800.0 PL=0
MOVL C01789 V=800.0 PL=0
MOVL C01790 V=800.0 PL=0
MOVL C01791 V=800.0 PL=0
MOVL C01792 V=800.0 PL=0
MOVL C01793 V=800.0 PL=0
MOVL C01794 V=800.0 PL=0
MOVL C01795 V=800.0 PL=0
MOVL C01796 V=800.0 PL=0
MOVL C01797 V=800.0 PL=0
MOVL C01798 V=800.0 PL=0
MOVL C01799 V=800.0 PL=0
MOVL C01800 V=800.0 PL=0
MOVL C01801 V=800.0 PL=0
MOVL C01802 V=800.0 PL=0
MOVL C01803 V=800.0 PL=0
MOVL C01804 V=800.0 PL=0
MOVL C01805 V=800.0 PL=0
MOVL C01806 V=800.0 PL=0
MOVL C01807 V=800.0 PL=0
MOVL C01808 V=800.0 PL=0
MOVL C01809 V=800.0 PL=0
MOVL C01810 V=800.0 PL=0
MOVL C01811 V=800.0 PL=0
MOVL C01812 V=800.0 PL=0
MOVL C01813 V=800.0 PL=0
MOVL C01814 V=800.0 PL=0
MOVL C01815 V=800.0 PL=0
MOVL C01816 V=800.0 PL=0
MOVL C01817 V=800.0 PL=0
MOVL C01818 V=800.0 PL=0
MOVL C01819 V=800.0 PL=0
MOVL C01820 V=800.0 PL=0
MOVL C01821 V=800.0 PL=0
MOVL C01822 V=800.0 PL=0
MOVL C01823 V=800.0 PL=0
MOVL C01824 V=800.0 PL=0
MOVL C01825 V=800.0 PL=0
MOVL C01826 V=800.0 PL=0
MOVL C01827 V=800.0 PL=0
MOVL C01828 V=800.0 PL=0
MOVL C01829 V=800.0 PL=0
MOVL C01830 V=800.0 PL=0
MOVL C01831 V=800.0 PL=0
MOVL C01832 V=800.0 PL=0
MOVL C01833 V=800.0 PL=0
MOVL C01834 V=800.0 PL=0
MOVL C01835 V=800.0 PL=0
MOVL C01836 V=800.0 PL=0
MOVL C01837 V=800.0 PL=0
MOVL C01838 V=800.0 PL=0
MOVL C01839 V=800.0 PL=0
MOVL C01840 V=800.0 PL=0
MOVL C01841 V=800.0 PL=0
MOVL C01842 V=800.0 PL=0
MOVL C01843 V=800.0 PL=0
MOVL C01844 V=800.0 PL=0
MOVL C01845 V=800.0 PL=0
MOVL C01846 V=800.0 PL=0
MOVL C01847 V=800.0 PL=0
MOVL C01848 V=800.0 PL=0
MOVL C01849 V=800.0 PL=0
MOVL C01850 V=800.0 PL=0
MOVL C01851 V=800.0 PL=0
MOVL C01852 V=800.0 PL=0
MOVL C01853 V=800.0 PL=0
MOVL C01854 V=800.0 PL=0
MOVL C01855 V=800.0 PL=0
MOVL C01856 V=800.0 PL=0
MOVL C01857 V=800.0 PL=0
MOVL C01858 V=800.0 PL=0
MOVL C01859 V=800.0 PL=0
MOVL C01860 V=800.0 PL=0
MOVL C01861 V=800.0 PL=0
MOVL C01862 V=800.0 PL=0
MOVL C01863 V=800.0 PL=0
MOVL C01864 V=800.0 PL=0
MOVL C01865 V=800.0 PL=0
MOVL C01866 V=800.0 PL=0
MOVL C01867 V=800.0 PL=0
MOVL C01868 V=800.0 PL=0
MOVL C01869 V=800.0 PL=0
MOVL C01870 V=800.0 PL=0
MOVL C01871 V=800.0 PL=0
MOVL C01872 V=800.0 PL=0
MOVL C01873 V=800.0 PL=0
MOVL C01874 V=800.0 PL=0
MOVL C01875 V=800.0 PL=0
MOVL C01876 V=800.0 PL=0
MOVL C01877 V=800.0 PL=0
MOVL C01878 V=800.0 PL=0
MOVL C01879 V=800.0 PL=0
MOVL C01880 V=800.0 PL=0
MOVL C01881 V=800.0 PL=0
MOVL C01882 V=800.0 PL=0
MOVL C01883 V=800.0 PL=0
MOVL C01884 V=800.0 PL=0
MOVL C01885 V=800.0 PL=0
MOVL C01886 V=800.0 PL=0
MOVL C01887 V=800.0 PL=0
MOVL C01888 V=800.0 PL=0
MOVL C01889 V=800.0 PL=0
MOVL C01890 V=800.0 PL=0
MOVL C01891 V=800.0 PL=0
MOVL C01892 V=800.0 PL=0
MOVL C01893 V=800.0 PL=0
MOVL C01894 V=800.0 PL=0
MOVL C01895 V=800.0 PL=0
MOVL C01896 V=800.0 PL=0
MOVL C01897 V=800.0 PL=0
MOVL C01898 V=800.0 PL=0
MOVL C01899 V=800.0 PL=0
MOVL C01900 V=800.0 PL=0
MOVL C01901 V=800.0 PL=0
MOVL C01902 V=800.0 PL=0
MOVL C01903 V=800.0 PL=0
MOVL C01904 V=800.0 PL=0
MOVL C01905 V=800.0 PL=0
MOVL C01906 V=800.0 PL=0
MOVL C01907 V=800.0 PL=0
MOVL C01908 V=800.0 PL=0
MOVL C01909 V=800.0 PL=0
MOVL C01910 V=800.0 PL=0
MOVL C01911 V=800.0 PL=0
MOVL C01912 V=800.0 PL=0
MOVL C01913 V=800.0 PL=0
MOVL C01914 V=800.0 PL=0
MOVL C01915 V=800.0 PL=0
MOVL C01916 V=800.0 PL=0
MOVL C01917 V=800.0 PL=0
MOVL C01918 V=800.0 PL=0
MOVL C01919 V=800.0 PL=0
MOVL C01920 V=800.0 PL=0
MOVL C01921 V=800.0 PL=0
MOVL C01922 V=800.0 PL=0
MOVL C01923 V=800.0 PL=0
MOVL C01924 V=800.0 PL=0
MOVL C01925 V=800.0 PL=0
MOVL C01926 V=800.0 PL=0
MOVL C01927 V=800.0 PL=0
MOVL C01928 V=800.0 PL=0
MOVL C01929 V=800.0 PL=0
MOVL C01930 V=800.0 PL=0
MOVL C01931 V=800.0 PL=0
MOVL C01932 V=800.0 PL=0
MOVL C01933 V=800.0 PL=0
MOVL C01934 V=800.0 PL=0
MOVL C01935 V=800.0 PL=0
MOVL C01936 V=800.0 PL=0
MOVL C01937 V=800.0 PL=0
MOVL C01938 V=800.0 PL=0
MOVL C01939 V=800.0 PL=0
MOVL C01940 V=800.0 PL=0
MOVL C01941 V=800.0 PL=0
MOVL C01942 V=800.0 PL=0
MOVL C01943 V=800.0 PL=0
MOVL C01944 V=800.0 PL=0
MOVL C01945 V=800.0 PL=0
MOVL C01946 V=800.0 PL=0
MOVL C01947 V=800.0 PL=0
MOVL C01948 V=800.0 PL=0
MOVL C01949 V=800.0 PL=0
MOVL C01950 V=800.0 PL=0
MOVL C01951 V=800.0 PL=0
MOVL C01952 V=800.0 PL=0
MOVL C01953 V=800.0 PL=0
MOVL C01954 V=800.0 PL=0
MOVL C01955 V=800.0 PL=0
MOVL C01956 V=800.0 PL=0
MOVL C01957 V=800.0 PL=0
MOVL C01958 V=800.0 PL=0
MOVL C01959 V=800.0 PL=0
MOVL C01960 V=800.0 PL=0
MOVL C01961 V=800.0 PL=0
MOVL C01962 V=800.0 PL=0
MOVL C01963 V=800.0 PL=0
MOVL C01964 V=800.0 PL=0
MOVL C01965 V=800.0 PL=0
MOVL C01966 V=800.0 PL=0
MOVL C01967 V=800.0 PL=0
MOVL C01968 V=800.0 PL=0
MOVL C01969 V=800.0 PL=0
MOVL C01970 V=800.0 PL=0
MOVL C01971 V=800.0 PL=0
MOVL C01972 V=800.0 PL=0
MOVL C01973 V=800.0 PL=0
MOVL C01974 V=800.0 PL=0
MOVL C01975 V=800.0 PL=0
MOVL C01976 V=800.0 PL=0
MOVL C01977 V=800.0 PL=0
MOVL C01978 V=800.0 PL=0
MOVL C01979 V=800.0 PL=0
MOVL C01980 V=800.0 PL=0
MOVL C01981 V=800.0 PL=0
MOVL C01982 V=800.0 PL=0
MOVL C01983 V=800.0 PL=0
MOVL C01984 V=800.0 PL=0
MOVL C01985 V=800.0 PL=0
MOVL C01986 V=800.0 PL=0
MOVL C01987 V=800.0 PL=0
MOVL C01988 V=800.0 PL=0
MOVL C01989 V=800.0 PL=0
MOVL C01990 V=800.0 PL=0
MOVL C01991 V=800.0 PL=0
MOVL C01992 V=800.0 PL=0
MOVL C01993 V=800.0 PL=0
MOVL C01994 V=800.0 PL=0
MOVL C01995 V=800.0 PL=0
MOVL C01996 V=800.0 PL=0
MOVL C01997 V=800.0 PL=0
MOVL C01998 V=800.0 PL=0
MOVL C01999 V=800.0 PL=0
MOVL C02000 V=800.0 PL=0
MOVL C02001 V=800.0 PL=0
MOVL C02002 V=800.0 PL=0
MOVL C02003 V=800.0 PL=0
MOVL C02004 V=800.0 PL=0
MOVL C02005 V=800.0 PL=0
MOVL C02006 V=800.0 PL=0
MOVL C02007 V=800.0 PL=0
MOVL C02008 V=800.0 PL=0
MOVL C02009 V=800.0 PL=0
MOVL C02010 V=800.0 PL=0
MOVL C02011 V=800.0 PL=0
MOVL C02012 V=800.0 PL=0
MOVL C02013 V=800.0 PL=0
MOVL C02014 V=800.0 PL=0
MOVL C02015 V=800.0 PL=0
MOVL C02016 V=800.0 PL=0
MOVL C02017 V=800.0 PL=0
MOVL C02018 V=800.0 PL=0
MOVL C02019 V=800.0 PL=0
MOVL C02020 V=800.0 PL=0
